(* CODESYS project LRF_2005_actual1.project
   Title: TemplateSPK1xxM01
   Version: 3.5.11.50
   Company: Production association OWEN

Project tree, tasks and I/O mapping:
  Device : SPK1xx[M01], Production association OWEN, order no. 7, version 3.5.11.57
    application Application
      libraries: Standard, * (System); CAA Memory, * (CAA Technical Workgroup); VisuDialogs, * (System); Standard64, * (System); VisuSymbols, 3.5.10.0 (System); Util, * (System)
      task OwenCloudTask (cyclic, interval T#100ms, priority 31) calls OwenStorage.CLOUD_PRG
      task MainTask (cyclic, interval t#10ms, priority 1) calls Main, Alarm, Motors
      task AlarmManagerTask (cyclic, interval 50 ms, priority 31) calls AlarmManager.Alarm_Prg
      task VISU_TASK (cyclic, interval 100 ms, priority 31) calls VisuElems.Visu_Prg
      Alarm Configuration
        alarm class Error (priority 10, acknowledge ACK_REP)
        alarm class Info (priority 100, acknowledge REP)
        alarm class Warning (priority 30, acknowledge REP)
        alarm group AlarmGroup
            11 [Error]: Comparison Equal, ExpressionToCompare TRUE, Expression GVL.SQ08_ALM - "Превышено время ожидания на переворот кантователя SQ08"
            21 [Error]: Comparison Equal, ExpressionToCompare TRUE, Expression GVL.M09UZ09_ALM - "Авария транспортера №5 M09UZ09"
            14 [Error]: Comparison Equal, ExpressionToCompare TRUE, Expression GVL.M01UZ01_ALM - "Авария дозатора обсыпного бункера M01UZ01"
            24 [Error]: Comparison Equal, ExpressionToCompare TRUE, Expression GVL.M14UZ14_ALM - "Авария транспортера №8 M14UZ14"
            19 [Error]: Comparison Equal, ExpressionToCompare TRUE, Expression GVL.M06UZ06_ALM - "Авария транспортера №3 M06UZ06"
            17 [Error]: Comparison Equal, ExpressionToCompare TRUE, Expression GVL.M04KM04_ALM - "Авария электромагнитного тормаза резчика M04KM04"
            12 [Info]: Comparison Equal, ExpressionToCompare TRUE, Expression GVL.XV01KV207_TSTOI - "Включен тестовый режим пресса "СЖАТЬ" XV01KV207"
            22 [Error]: Comparison Equal, ExpressionToCompare TRUE, Expression GVL.M11KM11_ALM - "Авария транспортера возврата песка №6 M11KM11"
            15 [Error]: Comparison Equal, ExpressionToCompare TRUE, Expression GVL.M02UZ02_ALM - "Авария резчика M02UZ02"
            25 [Error]: Comparison Equal, ExpressionToCompare TRUE, Expression GVL.A2_DI_SQ06_ALM - "Авария датчика верхнего положения выталкивателя SQ06 (геркон)."
            16 [Error]: Comparison Equal, ExpressionToCompare TRUE, Expression GVL.M03UZ03_ALM - "Авария транспортера №1 M03UZ03"
            10 [Error]: Comparison Equal, ExpressionToCompare TRUE, Expression GVL.M10KM10_ALM - "Авария маслостанции"
            20 [Error]: Comparison Equal, ExpressionToCompare TRUE, Expression GVL.M08KM08_ALM - "Авария транспортера подачи рамок №4 M08KM08"
            13 [Error]: Comparison Equal, ExpressionToCompare TRUE, Expression GVL.MV01KM00_ALM - "Авария вибратора обсыпного бункера MV01KM00"
            23 [Error]: Comparison Equal, ExpressionToCompare TRUE, Expression GVL.M12KM12_ALM - "Авария транспортера возврата обрези №7 M12KM12"
            18 [Error]: Comparison Equal, ExpressionToCompare TRUE, Expression GVL.M05UZ05_ALM - "Авария транспортера №2 M05UZ05"
            8 [Error]: Comparison Equal, ExpressionToCompare TRUE, Expression GVL.M07KM07_ALM - "Авария кантователя M07KM07"
            9 [Error]: Comparison Equal, ExpressionToCompare TRUE, Expression GVL.PI01_ALM - "Низкое давление масла PI01"
            0 [Error]: Comparison Equal, ExpressionToCompare FALSE, Expression GVL.A1_DI_SB_ALARM_STOP - "Нажата аварийная кнопка"
            1 [Error]: Comparison Equal, ExpressionToCompare TRUE, Expression GVL.A1_DI_QF25OK_ALM - "Отсутствует напряжение +24V QF25"
            2 [Error]: Comparison Equal, ExpressionToCompare TRUE, Expression GVL.A1_DI_QF26OK_ALM - "Отсутствует напряжение +24V QF26"
            3 [Error]: Comparison Equal, ExpressionToCompare TRUE, Expression GVL.A1_DI_380OK_ALM - "Отсутствует напряжение 380V QF1..QF16"
            4 [Error]: Comparison Equal, ExpressionToCompare TRUE, Expression GVL.XV01KV207_ALM - "Превышено время ожидания на сжатие пресса SQ05"
            5 [Error]: Comparison Equal, ExpressionToCompare TRUE, Expression GVL.XV02KV208_ALM - "Превышено время ожидания на разжатие пресса SQ04"
            6 [Error]: Comparison Equal, ExpressionToCompare TRUE, Expression GVL.XV03KV209_ALM - "Превышено время ожидания на выталкивание"
            7 [Error]: Comparison Equal, ExpressionToCompare TRUE, Expression GVL.XV04KV210_ALM - "Превышено время ожидания на возврат выталкивателя SQ06"
        text list AlarmGroup
        AlarmStorage
      global variables GVL
      visualisation TEST_FRAME_2
      program Motors [ST]
      visualisation SETTINGS_FRAME
      program SEQUENSER [ST]
      text list Mode
      visualisation PRF_FRAME
      TargetVariables/
        data type TRG_Drives
        data type TRG_Buzzer
        data type TRG_RTC
        global variables TargetVars
        data type TRG_Network
        data type TRG_Info
        data type TRG_Watchdog
        data type TRG_Debug
      visualisation ALARM_FRAME
      visualisation MODE_FRAME
      text list IM_TAGS
      visualisation TEST_FRAME_1
      visualisation Main
      program Alarm [ST]
      image pool Images
      program Main [ST]
      visualisation MAIN_FRAME
      text list IM
      visualisation MANUAL_FRAME_1
      global variables GVLR
      visualisation MANUAL_FRAME_2
      visualisation MANUAL_FRAME_3
    Info : Info, Production association OWEN, version 3.5.11.5003
        input  Application.TargetVars.stInfo.sVendorName : ARRAY [0..80] OF BYTE  // VENDOR
        input  Application.TargetVars.stInfo.sDeviceName : ARRAY [0..80] OF BYTE  // DEVICE
        input  Application.TargetVars.stInfo.sSerialId : ARRAY [0..80] OF BYTE  // SERIAL
        input  Application.TargetVars.stInfo.sRuntimeVersion : ARRAY [0..80] OF BYTE  // RUNTIME
        input  Application.TargetVars.stInfo.sFirmwareVersion : ARRAY [0..80] OF BYTE  // FIRMWARE
        input  Application.TargetVars.stInfo.sLinuxVersion : ARRAY [0..80] OF BYTE  // LINUX
        input  Application.TargetVars.stInfo.sNeedTargetVersion : ARRAY [0..80] OF BYTE  // TARGET
        input  Application.TargetVars.stInfo.sProjectName : ARRAY [0..80] OF BYTE  // PROJECT
        input  Application.TargetVars.stInfo.sAuthorName : ARRAY [0..80] OF BYTE  // AUTHOR
        input  Application.TargetVars.stInfo.sProjectVersion : ARRAY [0..80] OF BYTE  // VERSION
        input  Application.TargetVars.stInfo.sProjectProfile : ARRAY [0..80] OF BYTE  // PROFILE
        input  Application.TargetVars.stInfo.dtProjectLastChanges : DT  // LASTCHANGES
    Drives : Drives, Production association OWEN, version 3.5.11.5002
        input  Application.TargetVars.stDrives.uliFsFullSize : ULINT  // FS size
        input  Application.TargetVars.stDrives.uliFsUsedSize : ULINT  // FS used
        input  Application.TargetVars.stDrives.uliFsFreeSize : ULINT  // FS free
        input  Application.TargetVars.stDrives.xUsbMounted : BIT  // USB Mounted
        input  Application.TargetVars.stDrives.xUsbUnmountDone : BIT  // USB Unmount done
        input  Application.TargetVars.stDrives.uliUsbFullSize : ULINT  // USB size
        input  Application.TargetVars.stDrives.uliUsbUsedSize : ULINT  // USB used
        input  Application.TargetVars.stDrives.uliUsbFreeSize : ULINT  // USB free
        input  Application.TargetVars.stDrives.xSdMounted : BIT  // MMC Mounted
        input  Application.TargetVars.stDrives.xSdUnmountDone : BIT  // MMC Unmount done
        input  Application.TargetVars.stDrives.uliSdFullSize : ULINT  // MMC size
        input  Application.TargetVars.stDrives.uliSdUsedSize : ULINT  // MMC used
        input  Application.TargetVars.stDrives.uliSdFreeSize : ULINT  // MMC free
        output Application.TargetVars.stDrives.xEnable : BIT  // Enable Drives
        output Application.TargetVars.stDrives.xUsbUnmount : BIT  // USB Unmount
        output Application.TargetVars.stDrives.xSdUnmount : BIT  // MMC Unmount
    RS232_2 : Modbus COM, 3S - Smart Software Solutions GmbH, version 3.5.11.20
        settings: DataBits = 8; StopBits = 1; ComPort = 5
    OwenRTC : OwenRTC, Production association OWEN, version 3.5.11.5003
        input  Application.TargetVars.stRtc.uiGetYear : UINT  // Year
        input  Application.TargetVars.stRtc.usiGetMonth : USINT  // Month
        input  Application.TargetVars.stRtc.usiGetDay : USINT  // Day
        input  Application.TargetVars.stRtc.usiGetHour : USINT  // Hour
        input  Application.TargetVars.stRtc.usiGetMinute : USINT  // Minute
        input  Application.TargetVars.stRtc.usiGetSecond : USINT  // Second
        input  Application.TargetVars.stRtc.usiGetDayOfWeek : USINT  // Day of Week
        input  Application.TargetVars.stRtc.usiGetWeekOfYear : USINT  // Week of Year
        input  Application.GVL.PLC_DATE : ARRAY [0..80] OF BYTE  // Format Date
        input  Application.GVL.PLC_TIME : ARRAY [0..80] OF BYTE  // Format Time
        input  Application.TargetVars.stRtc.siGetUtcOffset : SINT  // UTC Offset
        input  Application.TargetVars.stRtc.xIsNtpEnabled : BIT  // NTP Enabled
        input  Application.TargetVars.stRtc.usiNtpErrorCode : USINT  // NTP Error
        input  Application.TargetVars.stRtc.ltSystemTick : LTIME  // System Timer
        input  Application.TargetVars.stRtc.dtDateAndTime : DT  // Date And Time
        output Application.TargetVars.stRtc.uiSetYear : UINT  // New Year
        output Application.TargetVars.stRtc.usiSetMonth : USINT  // New Month
        output Application.TargetVars.stRtc.usiSetDay : USINT  // New Day
        output Application.TargetVars.stRtc.usiSetHour : USINT  // New Hour
        output Application.TargetVars.stRtc.usiSetMinute : USINT  // New Minute
        output Application.TargetVars.stRtc.usiSetSecond : USINT  // New Second
        output Application.TargetVars.stRtc.siSetUtcOffset : SINT  // New UTC Offset
        output Application.TargetVars.stRtc.xUpdateSettings : BIT  // Set Settings DT
        output Application.TargetVars.stRtc.xEnableNtp : BIT  // Enable NTP
        output Application.TargetVars.stRtc.sPreferNtpServer : ARRAY [0..80] OF BYTE  // Prefer Server
    Debug : Debug, Production association OWEN, version 3.5.11.5002
        input  Application.TargetVars.stDebug.udiRamUsedSize : UDINT  // RAM used
        input  Application.TargetVars.stDebug.udiRamFreeSize : UDINT  // RAM free
        input  Application.TargetVars.stDebug.udiCountHandles : UDINT  // Open files
        input  Application.TargetVars.stDebug.udiProcUsage : UDINT  // Processor usage
        output Application.TargetVars.stDebug.xEnable : BIT  // Enable Debug
        output Application.TargetVars.stDebug.udiPollingTime : UDINT  // Debug pause
        unmapped channels: Core temp
    Watchdog : Watchdog, Production association OWEN, version 3.5.11.5003
        input  Application.TargetVars.stWatchdog.eHandlingType : INT  // Exception Handling
        input  Application.TargetVars.stWatchdog.udiLastExceptionCode : UDINT  // Last Exception Code
        input  Application.TargetVars.stWatchdog.sLastExceptionText : localTypes:STRING  // Last Exception Description
        input  Application.TargetVars.stWatchdog.dtLastExceptionTime : DT  // Last Exception Time
        input  Application.TargetVars.stWatchdog.xIsHardwareWatchdogReboot : BIT  // Hardware Watchdog Flag
        input  Application.TargetVars.stWatchdog.usiPowerRebootCount : USINT  // Power Reboot Count
        input  Application.TargetVars.stWatchdog.usiHardwareWatchdogRebootCount : USINT  // Watchdog Reboot Count
        input  Application.TargetVars.stWatchdog.usiExceptionRebootCount : USINT  // Exception Reboot Count
        input  Application.TargetVars.stWatchdog.usiCommandRebootCount : USINT  // Command Reboot Count
        output Application.TargetVars.stWatchdog.xDoReboot : BIT  // Reboot
        output Application.TargetVars.stWatchdog.xResetCounters : BIT  // Reset Counters
    Ethernet : Ethernet, 3S - Smart Software Solutions GmbH, version 3.5.11.0
        settings: IPAddress = [192,168,0,10]; SubnetMask = [255,255,0,0]; GatewayAddress = [192,168,0,1]; MACAddress = [16#E4,16#1E,16#0A,16#00,16#8E,16#B8]; NetworkInterfaceName = 'eth0'; NetworkInterfaceName = "eth0"; SaveCommunicationSettings = FALSE
      Modbus_TCP_Master : Modbus TCP Master, 3S - Smart Software Solutions GmbH, version 3.5.11.30
        A4 : MU210-410, Production association OWEN, version 3.5.11.6
            settings: IPAddress = [192, 168, 0, 6]
            input  Application.GVL.A4_DI_Modul_Fail : BIT  // Флаг ошибки
            output Application.GVL.A4_DO_HL02_32 : BOOL  // Битовая маска выходов (запись).Выход 1
            output Application.GVL.A4_DO_HL21 : BOOL  // Битовая маска выходов (запись).Выход 2
            output Application.GVL.A4_DO_HL35 : BOOL  // Битовая маска выходов (запись).Выход 3
            output Application.GVL.A4_DO_HL03_33 : BOOL  // Битовая маска выходов (запись).Выход 4
            output Application.GVL.A4_DO_HL04_34 : BOOL  // Битовая маска выходов (запись).Выход 5
            output Application.GVL.A4_DO_HL05 : BOOL  // Битовая маска выходов (запись).Выход 6
            output Application.GVL.A4_DO_XV01KV207 : BOOL  // Битовая маска выходов (запись).Выход 7
            output Application.GVL.A4_DO_XV02KV208 : BOOL  // Битовая маска выходов (запись).Выход 8
            output Application.GVL.A4_DO_XV03KV209 : BOOL  // Битовая маска выходов (запись).Выход 9
            output Application.GVL.A4_DO_XV04KV210 : BOOL  // Битовая маска выходов (запись).Выход 10
            output Application.GVL.A4_DO_XV05KV211 : BOOL  // Битовая маска выходов (запись).Выход 11
            output Application.GVL.A4_DO_XV06KV212 : BOOL  // Битовая маска выходов (запись).Выход 12
            output Application.GVL.A4_DO_RESERV01 : BOOL  // Битовая маска выходов (запись).Выход 13
            output Application.GVL.A4_DO_RESERV02 : BOOL  // Битовая маска выходов (запись).Выход 14
            output Application.GVL.A5_DO_M02UZ02_RUN_REV : BOOL  // Битовая маска выходов (запись).Выход 15
            output Application.GVL.A4_DO_RESERV04 : BOOL  // Битовая маска выходов (запись).Выход 16
            unmapped channels: Tmp, Исключить модуль из опроса, Битовая маска выходов (чтение), Битовая маска выходов (запись), Битовая маска диагностики выходов, Параметр ШИМ (чтение), Параметр ШИМ (чтение), Параметр ШИМ (чтение), Параметр ШИМ (чтение), Параметр ШИМ (чтение), Параметр ШИМ (чтение), Параметр ШИМ (чтение), Параметр ШИМ (чтение), Период ШИМ (чтение), Период ШИМ (чтение), Период ШИМ (чтение), Период ШИМ (чтение), Период ШИМ (чтение), Период ШИМ (чтение), Период ШИМ (чтение), Период ШИМ (чтение), Параметр ШИМ (запись), Параметр ШИМ (запись), Параметр ШИМ (запись), Параметр ШИМ (запись), Параметр ШИМ (запись), Параметр ШИМ (запись), Параметр ШИМ (запись), Параметр ШИМ (запись), Период ШИМ (запись), Период ШИМ (запись), Период ШИМ (запись), Период ШИМ (запись), Период ШИМ (запись), Период ШИМ (запись), Период ШИМ (запись), Период ШИМ (запись), Коэффициент заполнения ШИМ (чтение), Коэффициент заполнения ШИМ (чтение), Коэффициент заполнения ШИМ (чтение),
              Коэффициент заполнения ШИМ (чтение), Коэффициент заполнения ШИМ (чтение), Коэффициент заполнения ШИМ (чтение), Коэффициент заполнения ШИМ (чтение), Коэффициент заполнения ШИМ (чтение), Коэффициент заполнения ШИМ (чтение), Коэффициент заполнения ШИМ (чтение), Коэффициент заполнения ШИМ (чтение), Коэффициент заполнения ШИМ (чтение), Коэффициент заполнения ШИМ (чтение), Коэффициент заполнения ШИМ (чтение), Коэффициент заполнения ШИМ (чтение), Коэффициент заполнения ШИМ (чтение), Коэффициент заполнения ШИМ (запись), Коэффициент заполнения ШИМ (запись), Коэффициент заполнения ШИМ (запись), Коэффициент заполнения ШИМ (запись), Коэффициент заполнения ШИМ (запись), Коэффициент заполнения ШИМ (запись), Коэффициент заполнения ШИМ (запись), Коэффициент заполнения ШИМ (запись), Коэффициент заполнения ШИМ (запись), Коэффициент заполнения ШИМ (запись), Коэффициент заполнения ШИМ (запись), Коэффициент заполнения ШИМ (запись), Коэффициент заполнения ШИМ (запись), Коэффициент заполнения ШИМ (запись), Коэффициент заполнения ШИМ (запись), Коэффициент заполнения ШИМ (запись), Прочитать параметры, Записать параметры, Записать параметры, Записать параметры, Частота генератора (чтение), Частота генератора (чтение), Частота генератора (чтение), Частота генератора (запись), Частота генератора (запись), Частота генератора (запись), Количество импульсов генератора (чтение),
              Количество импульсов генератора (чтение), Количество импульсов генератора (чтение), Количество импульсов генератора (запись), Количество импульсов генератора (запись), Количество импульсов генератора (запись), Осталось сгенерировать импульсов, Осталось сгенерировать импульсов, Осталось сгенерировать импульсов
        A1 : MV210-202, Production association OWEN, version 3.5.11.6
            settings: IPAddress = [192, 168, 0, 3]
            input  Application.GVL.A1_DI_Modul_Fail : BIT  // Флаг ошибки
            input  Application.GVL.A1_DI_QF25OK : BOOL  // Битовая маска входов.Вход 1
            input  Application.GVL.A1_DI_QF26OK : BOOL  // Битовая маска входов.Вход 2
            input  Application.GVL.A1_DI_380OK : BOOL  // Битовая маска входов.Вход 3
            input  Application.GVL.A1_DI_SB_ALARM_STOP : BOOL  // Битовая маска входов.Вход 4
            input  Application.GVL.A1_DI_SB_STOP : BOOL  // Битовая маска входов.Вход 5
            input  Application.GVL.A1_DI_SB_1st_OPER : BOOL  // Битовая маска входов.Вход 6
            input  Application.GVL.A1_DI_SB_2nd_OPER : BOOL  // Битовая маска входов.Вход 7
            input  Application.GVL.A1_DI_SB_RESET : BOOL  // Битовая маска входов.Вход 8
            input  Application.GVL.A1_DI_SB_START : BOOL  // Битовая маска входов.Вход 9
            input  Application.GVL.A1_DI_SA01 : BOOL  // Битовая маска входов.Вход 10
            input  Application.GVL.A1_DI_SB_TEST : BOOL  // Битовая маска входов.Вход 11
            input  Application.GVL.A1_DI_MV01KM00_ON : BOOL  // Битовая маска входов.Вход 12
            input  Application.GVL.A1_DI_M01UZ01_ON : BOOL  // Битовая маска входов.Вход 13
            input  Application.GVL.A1_DI_RESERV01 : BOOL  // Битовая маска входов.Вход 14
            input  Application.GVL.A1_DI_M03UZ03_ON : BOOL  // Битовая маска входов.Вход 15
            input  Application.GVL.A1_DI_M04KM04_ON : BOOL  // Битовая маска входов.Вход 16
            input  Application.GVL.A1_DI_M05UZ05_ON : BOOL  // Битовая маска входов.Вход 17
            input  Application.GVL.A1_DI_M06UZ06_ON : BOOL  // Битовая маска входов.Вход 18
            input  Application.GVL.A1_DI_M07KM07_ON : BOOL  // Битовая маска входов.Вход 19
            input  Application.GVL.A1_DI_M08KM08_ON : BOOL  // Битовая маска входов.Вход 20
            unmapped channels: Tmp, Исключить модуль из опроса, Битовая маска входов, Значение, Значение, Значение, Значение, Значение, Значение, Значение, Значение, Значение счетчика, Значение счетчика, Значение счетчика, Значение счетчика, Значение счетчика, Значение счетчика, Значение счетчика, Значение счетчика, Значение счетчика, Значение счетчика, Значение счетчика, Значение счетчика, Сбросить значение, Сбросить значение, Сбросить значение, Сбросить значение, Сбросить значение, Сбросить значение, Сбросить значение, Сбросить значение, Сбросить счетчик, Сбросить счетчик, Сбросить счетчик, Сбросить счетчик, Сбросить счетчик, Сбросить счетчик, Сбросить счетчик, Сбросить счетчик, Сбросить счетчик,
              Сбросить счетчик, Сбросить счетчик, Сбросить счетчик
        A5 : MU210-410, Production association OWEN, version 3.5.11.6
            settings: IPAddress = [192, 168, 0, 7]
            input  Application.GVL.A5_DI_Modul_Fail : BIT  // Флаг ошибки
            output Application.GVL.A5_DO_MV01KM00_RUN : BOOL  // Битовая маска выходов (запись).Выход 1
            output Application.GVL.A5_DO_M01UZ01_RUN : BOOL  // Битовая маска выходов (запись).Выход 2
            output Application.GVL.A5_DO_M02UZ02_RUN_FORW : BOOL  // Битовая маска выходов (запись).Выход 3
            output Application.GVL.A5_DO_M03UZ03_RUN : BOOL  // Битовая маска выходов (запись).Выход 4
            output Application.GVL.A5_DO_M04KM04_RUN : BOOL  // Битовая маска выходов (запись).Выход 5
            output Application.GVL.A5_DO_M05UZ05_RUN : BOOL  // Битовая маска выходов (запись).Выход 6
            output Application.GVL.A5_DO_M06UZ06_RUN : BOOL  // Битовая маска выходов (запись).Выход 7
            output Application.GVL.A5_DO_M07KM07_RUN : BOOL  // Битовая маска выходов (запись).Выход 8
            output Application.GVL.A5_DO_M08KM08_RUN : BOOL  // Битовая маска выходов (запись).Выход 9
            output Application.GVL.A5_DO_M09UZ09_RUN : BOOL  // Битовая маска выходов (запись).Выход 10
            output Application.GVL.A5_DO_M10KM10_RUN : BOOL  // Битовая маска выходов (запись).Выход 11
            output Application.GVL.A5_DO_M11KM11_RUN : BOOL  // Битовая маска выходов (запись).Выход 12
            output Application.GVL.A5_DO_M12KM12_RUN : BOOL  // Битовая маска выходов (запись).Выход 13
            output Application.GVL.A5_DO_M13KM13_RUN : BOOL  // Битовая маска выходов (запись).Выход 14
            output Application.GVL.A5_DO_M14UZ14_RUN : BOOL  // Битовая маска выходов (запись).Выход 15
            output Application.GVL.A5_DO_RESERV01 : BOOL  // Битовая маска выходов (запись).Выход 16
            unmapped channels: Tmp, Исключить модуль из опроса, Битовая маска выходов (чтение), Битовая маска выходов (запись), Битовая маска диагностики выходов, Параметр ШИМ (чтение), Параметр ШИМ (чтение), Параметр ШИМ (чтение), Параметр ШИМ (чтение), Параметр ШИМ (чтение), Параметр ШИМ (чтение), Параметр ШИМ (чтение), Параметр ШИМ (чтение), Период ШИМ (чтение), Период ШИМ (чтение), Период ШИМ (чтение), Период ШИМ (чтение), Период ШИМ (чтение), Период ШИМ (чтение), Период ШИМ (чтение), Период ШИМ (чтение), Параметр ШИМ (запись), Параметр ШИМ (запись), Параметр ШИМ (запись), Параметр ШИМ (запись), Параметр ШИМ (запись), Параметр ШИМ (запись), Параметр ШИМ (запись), Параметр ШИМ (запись), Период ШИМ (запись), Период ШИМ (запись), Период ШИМ (запись), Период ШИМ (запись), Период ШИМ (запись), Период ШИМ (запись), Период ШИМ (запись), Период ШИМ (запись), Коэффициент заполнения ШИМ (чтение), Коэффициент заполнения ШИМ (чтение), Коэффициент заполнения ШИМ (чтение),
              Коэффициент заполнения ШИМ (чтение), Коэффициент заполнения ШИМ (чтение), Коэффициент заполнения ШИМ (чтение), Коэффициент заполнения ШИМ (чтение), Коэффициент заполнения ШИМ (чтение), Коэффициент заполнения ШИМ (чтение), Коэффициент заполнения ШИМ (чтение), Коэффициент заполнения ШИМ (чтение), Коэффициент заполнения ШИМ (чтение), Коэффициент заполнения ШИМ (чтение), Коэффициент заполнения ШИМ (чтение), Коэффициент заполнения ШИМ (чтение), Коэффициент заполнения ШИМ (чтение), Коэффициент заполнения ШИМ (запись), Коэффициент заполнения ШИМ (запись), Коэффициент заполнения ШИМ (запись), Коэффициент заполнения ШИМ (запись), Коэффициент заполнения ШИМ (запись), Коэффициент заполнения ШИМ (запись), Коэффициент заполнения ШИМ (запись), Коэффициент заполнения ШИМ (запись), Коэффициент заполнения ШИМ (запись), Коэффициент заполнения ШИМ (запись), Коэффициент заполнения ШИМ (запись), Коэффициент заполнения ШИМ (запись), Коэффициент заполнения ШИМ (запись), Коэффициент заполнения ШИМ (запись), Коэффициент заполнения ШИМ (запись), Коэффициент заполнения ШИМ (запись), Прочитать параметры, Записать параметры, Записать параметры, Записать параметры, Частота генератора (чтение), Частота генератора (чтение), Частота генератора (чтение), Частота генератора (запись), Частота генератора (запись), Частота генератора (запись), Количество импульсов генератора (чтение),
              Количество импульсов генератора (чтение), Количество импульсов генератора (чтение), Количество импульсов генератора (запись), Количество импульсов генератора (запись), Количество импульсов генератора (запись), Осталось сгенерировать импульсов, Осталось сгенерировать импульсов, Осталось сгенерировать импульсов
        A3 : MK210-302, Production association OWEN, version 3.5.11.6
            settings: IPAddress = [192, 168, 0, 5]
            input  Application.GVL.A3_DI_Modul_Fail : BIT  // Флаг ошибки
            input  Application.GVL.A3_DI_SQ10 : BOOL  // Битовая маска входов.Вход 1
            input  Application.GVL.A3_DI_SQ13 : BOOL  // Битовая маска входов.Вход 2
            input  Application.GVL.A3_DI_SQ14 : BOOL  // Битовая маска входов.Вход 3
            input  Application.GVL.A3_DI_RESERV01 : BOOL  // Битовая маска входов.Вход 4
            input  Application.GVL.A3_DI_SQ11 : BOOL  // Битовая маска входов.Вход 5
            input  Application.GVL.A3_DI_SQ12 : BOOL  // Битовая маска входов.Вход 6
            input  Application.GVL.A3_DI_RESERV02 : BOOL  // Битовая маска входов.Вход 7
            input  Application.GVL.A3_DI_KV301 : BOOL  // Битовая маска входов.Вход 8
            input  Application.GVL.A3_DI_KV302 : BOOL  // Битовая маска входов.Вход 9
            input  Application.GVL.A3_DI_PI01 : BOOL  // Битовая маска входов.Вход 10
            input  Application.GVL.A3_DI_RESERV03 : BOOL  // Битовая маска входов.Вход 11
            input  Application.GVL.A3_DI_RESERV04 : BOOL  // Битовая маска входов.Вход 12
            output Application.GVL.A3_DO_KV303 : BOOL  // Битовая маска выходов (запись).Выход 1
            output Application.GVL.A3_DO_KV304 : BOOL  // Битовая маска выходов (запись).Выход 2
            output Application.GVL.A3_DO_RESERV01 : BOOL  // Битовая маска выходов (запись).Выход 3
            output Application.GVL.A3_DO_RESERV02 : BOOL  // Битовая маска выходов (запись).Выход 4
            unmapped channels: Tmp, Исключить модуль из опроса, Битовая маска входов, Значение счетчика, Значение счетчика, Значение счетчика, Значение счетчика, Значение счетчика, Значение счетчика, Значение счетчика, Значение счетчика, Значение счетчика, Значение счетчика, Значение счетчика, Значение счетчика, Битовая маска выходов (чтение), Битовая маска выходов (запись), Сбросить счетчик, Сбросить счетчик, Сбросить счетчик, Сбросить счетчик, Сбросить счетчик, Сбросить счетчик, Сбросить счетчик, Сбросить счетчик, Сбросить счетчик, Сбросить счетчик, Сбросить счетчик, Сбросить счетчик, Период ШИМ (чтение), Период ШИМ (чтение), Период ШИМ (чтение), Период ШИМ (чтение), Период ШИМ (запись), Период ШИМ (запись), Период ШИМ (запись), Период ШИМ (запись), Коэффициент заполнения ШИМ (чтение), Коэффициент заполнения ШИМ (чтение), Коэффициент заполнения ШИМ (чтение),
              Коэффициент заполнения ШИМ (чтение), Коэффициент заполнения ШИМ (запись), Коэффициент заполнения ШИМ (запись), Коэффициент заполнения ШИМ (запись), Коэффициент заполнения ШИМ (запись)
        A2 : MV210-202, Production association OWEN, version 3.5.11.6
            settings: IPAddress = [192, 168, 0, 4]
            input  Application.GVL.A2_DI_Modul_Fail : BIT  // Флаг ошибки
            input  Application.GVL.A2_DI_M09UZ09_ON : BOOL  // Битовая маска входов.Вход 1
            input  Application.GVL.A2_DI_M10KM10_ON : BOOL  // Битовая маска входов.Вход 2
            input  Application.GVL.A2_DI_M11KM11_ON : BOOL  // Битовая маска входов.Вход 3
            input  Application.GVL.A2_DI_M12KM12_ON : BOOL  // Битовая маска входов.Вход 4
            input  Application.GVL.A2_DI_M13KM13_ON : BOOL  // Битовая маска входов.Вход 5
            input  Application.GVL.A2_DI_M14UZ14_ON : BOOL  // Битовая маска входов.Вход 6
            input  Application.GVL.A2_DI_SQ01 : BOOL  // Битовая маска входов.Вход 7
            input  Application.GVL.A2_DI_SQ02 : BOOL  // Битовая маска входов.Вход 8
            input  Application.GVL.A2_DI_SQ15 : BOOL  // Битовая маска входов.Вход 9
            input  Application.GVL.A2_DI_SQ03 : BOOL  // Битовая маска входов.Вход 10
            input  Application.GVL.A2_DI_RESERV02 : BOOL  // Битовая маска входов.Вход 11
            input  Application.GVL.A2_DI_SQ04 : BOOL  // Битовая маска входов.Вход 12
            input  Application.GVL.A2_DI_SQ05 : BOOL  // Битовая маска входов.Вход 13
            input  Application.GVL.A2_DI_SQ06 : BOOL  // Битовая маска входов.Вход 14
            input  Application.GVL.A2_DI_SQ07 : BOOL  // Битовая маска входов.Вход 15
            input  Application.GVL.A2_DI_SQ08 : BOOL  // Битовая маска входов.Вход 16
            input  Application.GVL.A2_DI_RESERV03 : BOOL  // Битовая маска входов.Вход 17
            input  Application.GVL.A2_DI_RESERV04 : BOOL  // Битовая маска входов.Вход 18
            input  Application.GVL.A2_DI_RESERV05 : BOOL  // Битовая маска входов.Вход 19
            input  Application.GVL.A2_DI_SQ09 : BOOL  // Битовая маска входов.Вход 20
            input  Application.GVL.A2_DI_SQ02_CNT : UDINT  // Значение
            input  Application.GVL.A2_DI_SQ08_CNT : UDINT  // Значение счетчика
            output Application.GVL.RESET_SQ2_CNT : BIT  // Сбросить значение
            output Application.GVL.RESET_CNT : BIT  // Сбросить счетчик
            unmapped channels: Tmp, Исключить модуль из опроса, Битовая маска входов, Значение, Значение, Значение, Значение, Значение, Значение, Значение, Значение счетчика, Значение счетчика, Значение счетчика, Значение счетчика, Значение счетчика, Значение счетчика, Значение счетчика, Значение счетчика, Значение счетчика, Значение счетчика, Значение счетчика, Сбросить значение, Сбросить значение, Сбросить значение, Сбросить значение, Сбросить значение, Сбросить значение, Сбросить значение, Сбросить счетчик, Сбросить счетчик, Сбросить счетчик, Сбросить счетчик, Сбросить счетчик, Сбросить счетчик, Сбросить счетчик, Сбросить счетчик, Сбросить счетчик, Сбросить счетчик, Сбросить счетчик
    RS485_2 : Modbus COM, 3S - Smart Software Solutions GmbH, version 3.5.11.20
        settings: DataBits = 8; StopBits = 1; ComPort = 2
    RS485_3 : Modbus COM, 3S - Smart Software Solutions GmbH, version 3.5.11.20
        settings: DataBits = 8; StopBits = 1; ComPort = 3
    RS232_1 : Modbus COM, 3S - Smart Software Solutions GmbH, version 3.5.11.20
        settings: DataBits = 8; StopBits = 1; ComPort = 4
    RS485_1 : Modbus COM, 3S - Smart Software Solutions GmbH, version 3.5.11.20
        settings: DataBits = 8; StopBits = 1; ComPort = 1
      Modbus_Master_COM_Port_1 : Modbus Master, COM Port, 3S - Smart Software Solutions GmbH, version 3.5.11.20
        UZ06 : Modbus Slave, COM Port, 3S - Smart Software Solutions GmbH, version 3.5.10.30
            settings: SlaveAddress = 6; ResponseTimeout = 1000; UseExtendedFunctionCodes = TRUE; UZ_FREQUENCY_PV.Function Code = 3; UZ_FREQUENCY_PV.Read Offset = 16#C421; UZ_FREQUENCY_PV.Read Length = 1; UZ_FREQUENCY_PV.Write Offset = 0; UZ_FREQUENCY_PV.Write Length = 0; UZ_FREQUENCY_PV.Cycle Time = 100; UZ_STATUS.Function Code = 3; UZ_STATUS.Read Offset = 16#C417; UZ_STATUS.Read Length = 1; UZ_STATUS.Write Offset = 0; UZ_STATUS.Write Length = 0; UZ_STATUS.Cycle Time = 100; UZ_CONTROL.Function Code = 6; UZ_CONTROL.Read Offset = 0; UZ_CONTROL.Read Length = 0; UZ_CONTROL.Write Offset = 16#C34F; UZ_CONTROL.Write Length = 1; UZ_CONTROL.Cycle Time = 100; UZ_FREQUENCY_SP.Function Code = 6; UZ_FREQUENCY_SP.Read Offset = 0; UZ_FREQUENCY_SP.Read Length = 0; UZ_FREQUENCY_SP.Write Offset = 16#C359; UZ_FREQUENCY_SP.Write Length = 1; UZ_FREQUENCY_SP.Cycle Time = 100
            input  Application.GVL.UZ06_Freq_PV : ARRAY[0..0] OF WORD  // UZ_FREQUENCY_PV
            output Application.GVL.UZ06_Freq_SP : ARRAY[0..0] OF WORD  // UZ_FREQUENCY_SP
            unmapped channels: UZ_STATUS, UZ_CONTROL
        UZ03 : Modbus Slave, COM Port, 3S - Smart Software Solutions GmbH, version 3.5.10.30
            settings: SlaveAddress = 3; ResponseTimeout = 1000; UseExtendedFunctionCodes = TRUE; UZ_FREQUENCY_PV.Function Code = 3; UZ_FREQUENCY_PV.Read Offset = 16#C421; UZ_FREQUENCY_PV.Read Length = 1; UZ_FREQUENCY_PV.Write Offset = 0; UZ_FREQUENCY_PV.Write Length = 0; UZ_FREQUENCY_PV.Cycle Time = 100; UZ_STATUS.Function Code = 3; UZ_STATUS.Read Offset = 16#C417; UZ_STATUS.Read Length = 1; UZ_STATUS.Write Offset = 0; UZ_STATUS.Write Length = 0; UZ_STATUS.Cycle Time = 100; UZ_CONTROL.Function Code = 6; UZ_CONTROL.Read Offset = 0; UZ_CONTROL.Read Length = 0; UZ_CONTROL.Write Offset = 16#C34F; UZ_CONTROL.Write Length = 1; UZ_CONTROL.Cycle Time = 100; UZ_FREQUENCY_SP.Function Code = 6; UZ_FREQUENCY_SP.Read Offset = 0; UZ_FREQUENCY_SP.Read Length = 0; UZ_FREQUENCY_SP.Write Offset = 16#C359; UZ_FREQUENCY_SP.Write Length = 1; UZ_FREQUENCY_SP.Cycle Time = 100
            input  Application.GVL.UZ03_Freq_PV : ARRAY[0..0] OF WORD  // UZ_FREQUENCY_PV
            input  Application.GVL.UZ03_Status_Word : ARRAY[0..0] OF WORD  // UZ_STATUS
            output Application.GVL.UZ03_Freq_SP : ARRAY[0..0] OF WORD  // UZ_FREQUENCY_SP
            unmapped channels: UZ_CONTROL
        UZ05 : Modbus Slave, COM Port, 3S - Smart Software Solutions GmbH, version 3.5.10.30
            settings: SlaveAddress = 5; ResponseTimeout = 1000; UseExtendedFunctionCodes = TRUE; UZ_FREQUENCY_PV.Function Code = 3; UZ_FREQUENCY_PV.Read Offset = 16#C421; UZ_FREQUENCY_PV.Read Length = 1; UZ_FREQUENCY_PV.Write Offset = 0; UZ_FREQUENCY_PV.Write Length = 0; UZ_FREQUENCY_PV.Cycle Time = 100; UZ_STATUS.Function Code = 3; UZ_STATUS.Read Offset = 16#C417; UZ_STATUS.Read Length = 1; UZ_STATUS.Write Offset = 0; UZ_STATUS.Write Length = 0; UZ_STATUS.Cycle Time = 100; UZ_CONTROL.Function Code = 6; UZ_CONTROL.Read Offset = 0; UZ_CONTROL.Read Length = 0; UZ_CONTROL.Write Offset = 16#C34F; UZ_CONTROL.Write Length = 1; UZ_CONTROL.Cycle Time = 100; UZ_FREQUENCY_SP.Function Code = 6; UZ_FREQUENCY_SP.Read Offset = 0; UZ_FREQUENCY_SP.Read Length = 0; UZ_FREQUENCY_SP.Write Offset = 16#C359; UZ_FREQUENCY_SP.Write Length = 1; UZ_FREQUENCY_SP.Cycle Time = 100
            input  Application.GVL.UZ05_Freq_PV : ARRAY[0..0] OF WORD  // UZ_FREQUENCY_PV
            output Application.GVL.UZ05_Freq_SP : ARRAY[0..0] OF WORD  // UZ_FREQUENCY_SP
            unmapped channels: UZ_STATUS, UZ_CONTROL
        UZ09 : Modbus Slave, COM Port, 3S - Smart Software Solutions GmbH, version 3.5.10.30
            settings: SlaveAddress = 9; ResponseTimeout = 1000; UseExtendedFunctionCodes = TRUE; UZ_FREQUENCY_PV.Function Code = 3; UZ_FREQUENCY_PV.Read Offset = 16#C421; UZ_FREQUENCY_PV.Read Length = 1; UZ_FREQUENCY_PV.Write Offset = 0; UZ_FREQUENCY_PV.Write Length = 0; UZ_FREQUENCY_PV.Cycle Time = 100; UZ_STATUS.Function Code = 3; UZ_STATUS.Read Offset = 16#C417; UZ_STATUS.Read Length = 1; UZ_STATUS.Write Offset = 0; UZ_STATUS.Write Length = 0; UZ_STATUS.Cycle Time = 100; UZ_CONTROL.Function Code = 6; UZ_CONTROL.Read Offset = 0; UZ_CONTROL.Read Length = 0; UZ_CONTROL.Write Offset = 16#C34F; UZ_CONTROL.Write Length = 1; UZ_CONTROL.Cycle Time = 100; UZ_FREQUENCY_SP.Function Code = 6; UZ_FREQUENCY_SP.Read Offset = 0; UZ_FREQUENCY_SP.Read Length = 0; UZ_FREQUENCY_SP.Write Offset = 16#C359; UZ_FREQUENCY_SP.Write Length = 1; UZ_FREQUENCY_SP.Cycle Time = 100
            input  Application.GVL.UZ09_Freq_PV : ARRAY[0..0] OF WORD  // UZ_FREQUENCY_PV
            output Application.GVL.UZ09_Freq_SP : ARRAY[0..0] OF WORD  // UZ_FREQUENCY_SP
            unmapped channels: UZ_STATUS, UZ_CONTROL
        UZ02 : Modbus Slave, COM Port, 3S - Smart Software Solutions GmbH, version 3.5.10.30
            settings: SlaveAddress = 2; ResponseTimeout = 1000; UseExtendedFunctionCodes = TRUE; UZ_FREQUENCY_PV.Function Code = 3; UZ_FREQUENCY_PV.Read Offset = 16#C421; UZ_FREQUENCY_PV.Read Length = 1; UZ_FREQUENCY_PV.Write Offset = 0; UZ_FREQUENCY_PV.Write Length = 0; UZ_FREQUENCY_PV.Cycle Time = 100; UZ_STATUS.Function Code = 3; UZ_STATUS.Read Offset = 16#C417; UZ_STATUS.Read Length = 1; UZ_STATUS.Write Offset = 0; UZ_STATUS.Write Length = 0; UZ_STATUS.Cycle Time = 100; UZ_CONTROL.Function Code = 6; UZ_CONTROL.Read Offset = 0; UZ_CONTROL.Read Length = 0; UZ_CONTROL.Write Offset = 16#C34F; UZ_CONTROL.Write Length = 1; UZ_CONTROL.Cycle Time = 100; UZ_FREQUENCY_SP.Function Code = 6; UZ_FREQUENCY_SP.Read Offset = 0; UZ_FREQUENCY_SP.Read Length = 0; UZ_FREQUENCY_SP.Write Offset = 16#C359; UZ_FREQUENCY_SP.Write Length = 1; UZ_FREQUENCY_SP.Cycle Time = 100
            input  Application.GVL.UZ02_Freq_PV : ARRAY[0..0] OF WORD  // UZ_FREQUENCY_PV
            input  Application.GVL.UZ02_Status_Word : ARRAY[0..0] OF WORD  // UZ_STATUS
            output Application.GVL.UZ02_Freq_SP : ARRAY[0..0] OF WORD  // UZ_FREQUENCY_SP
            unmapped channels: UZ_CONTROL
        UZ01 : Modbus Slave, COM Port, 3S - Smart Software Solutions GmbH, version 3.5.10.30
            settings: SlaveAddress = 1; ResponseTimeout = 1000; UseExtendedFunctionCodes = TRUE; UZ_FREQUENCY_PV.Function Code = 3; UZ_FREQUENCY_PV.Read Offset = 16#C421; UZ_FREQUENCY_PV.Read Length = 1; UZ_FREQUENCY_PV.Write Offset = 0; UZ_FREQUENCY_PV.Write Length = 0; UZ_FREQUENCY_PV.Cycle Time = 100; UZ_STATUS.Function Code = 3; UZ_STATUS.Read Offset = 16#C417; UZ_STATUS.Read Length = 1; UZ_STATUS.Write Offset = 0; UZ_STATUS.Write Length = 0; UZ_STATUS.Cycle Time = 100; UZ_CONTROL.Function Code = 6; UZ_CONTROL.Read Offset = 0; UZ_CONTROL.Read Length = 0; UZ_CONTROL.Write Offset = 16#C34F; UZ_CONTROL.Write Length = 1; UZ_CONTROL.Cycle Time = 100; UZ_FREQUENCY_SP.Function Code = 6; UZ_FREQUENCY_SP.Read Offset = 0; UZ_FREQUENCY_SP.Read Length = 0; UZ_FREQUENCY_SP.Write Offset = 16#C359; UZ_FREQUENCY_SP.Write Length = 1; UZ_FREQUENCY_SP.Cycle Time = 100
            input  Application.GVL.UZ01_Freq_PV : ARRAY[0..0] OF WORD  // UZ_FREQUENCY_PV
            input  Application.GVL.UZ01_Status_Word : ARRAY[0..0] OF WORD  // UZ_STATUS
            output Application.GVL.UZ01_Freq_SP : ARRAY[0..0] OF WORD  // UZ_FREQUENCY_SP
            unmapped channels: UZ_CONTROL
        UZ14 : Modbus Slave, COM Port, 3S - Smart Software Solutions GmbH, version 3.5.10.30
            settings: SlaveAddress = 14; ResponseTimeout = 1000; UseExtendedFunctionCodes = TRUE; UZ_FREQUENCY_PV.Function Code = 3; UZ_FREQUENCY_PV.Read Offset = 16#C421; UZ_FREQUENCY_PV.Read Length = 1; UZ_FREQUENCY_PV.Write Offset = 0; UZ_FREQUENCY_PV.Write Length = 0; UZ_FREQUENCY_PV.Cycle Time = 100; UZ_STATUS.Function Code = 3; UZ_STATUS.Read Offset = 16#C417; UZ_STATUS.Read Length = 1; UZ_STATUS.Write Offset = 0; UZ_STATUS.Write Length = 0; UZ_STATUS.Cycle Time = 100; UZ_CONTROL.Function Code = 6; UZ_CONTROL.Read Offset = 0; UZ_CONTROL.Read Length = 0; UZ_CONTROL.Write Offset = 16#C34F; UZ_CONTROL.Write Length = 1; UZ_CONTROL.Cycle Time = 100; UZ_FREQUENCY_SP.Function Code = 6; UZ_FREQUENCY_SP.Read Offset = 0; UZ_FREQUENCY_SP.Read Length = 0; UZ_FREQUENCY_SP.Write Offset = 16#C359; UZ_FREQUENCY_SP.Write Length = 1; UZ_FREQUENCY_SP.Cycle Time = 100
            input  Application.GVL.UZ14_Freq_PV : ARRAY[0..0] OF WORD  // UZ_FREQUENCY_PV
            output Application.GVL.UZ14_Freq_SP : ARRAY[0..0] OF WORD  // UZ_FREQUENCY_SP
            unmapped channels: UZ_STATUS, UZ_CONTROL
    Screen : Screen, Production association OWEN, version 3.5.11.5002
        unmapped channels: Get Brightness, Dim time, Off time, Full brightness, Dim brightness, Off brightness, Dim visu name, Off visu name, On visu name, Wake up
    Network : Network, Production association OWEN, version 3.5.11.5002
        input  Application.TargetVars.stNetwork.xGetDhcp : BIT  // DHCP enabled
        input  Application.TargetVars.stNetwork.abyGetIp : ARRAY [0..3] OF BYTE  // IP
        input  Application.TargetVars.stNetwork.abyGetMask : ARRAY [0..3] OF BYTE  // Mask
        input  Application.TargetVars.stNetwork.abyGetGateway : ARRAY [0..3] OF BYTE  // Gateway
        input  Application.TargetVars.stNetwork.abyGetMac : ARRAY [0..5] OF BYTE  // MAC
        input  Application.TargetVars.stNetwork.sGetHostname : ARRAY [0..80] OF BYTE  // Hostname
        output Application.TargetVars.stNetwork.xSetDhcp : BIT  // Enable DHCP
        output Application.TargetVars.stNetwork.abySetIp : ARRAY [0..3] OF BYTE  // New IP
        output Application.TargetVars.stNetwork.abySetMask : ARRAY [0..3] OF BYTE  // New Mask
        output Application.TargetVars.stNetwork.abySetGateway : ARRAY [0..3] OF BYTE  // New Gateway
        output Application.TargetVars.stNetwork.sSetHostname : ARRAY [0..80] OF BYTE  // New Hostname
        output Application.TargetVars.stNetwork.xSetSettings : BIT  // Set Settings
    Buzzer : Buzzer, Production association OWEN, version 3.5.11.5002
        input  Application.TargetVars.stBuzzer.xGet : BIT  // Buzzer enabled
        output Application.TargetVars.stBuzzer.xSet : BIT  // Enable Buzzer
    OwenCloud : OwenCloud, Production association OWEN, version 3.5.11.5003
        unmapped channels: OwenCloud enabled, Folder error, Symbol error, Enable OwenCloud
  libraries: VisuSymbols, 3.5.10.0 (System)
  5ce3da45-db07-42e7-a21c-a00fff4ed8f6|Ленин - для мнемосхем\2-огр. паллет вверху.png
  5ce3da45-db07-42e7-a21c-a00fff4ed8f6|C:\Users\Alex\Desktop\LRF\IMG\M03UZ03_ON.png
  5ce3da45-db07-42e7-a21c-a00fff4ed8f6|Ленин - для мнемосхем\2-Подложка.png
  5ce3da45-db07-42e7-a21c-a00fff4ed8f6|C:\Users\Alex\Desktop\LRF\IMG\SQ04.png
  5ce3da45-db07-42e7-a21c-a00fff4ed8f6|Ленин - для мнемосхем\RUN-тр-р угловой.png
  5ce3da45-db07-42e7-a21c-a00fff4ed8f6|C:\Users\Alex\Desktop\LRF\IMG\M12KM12_ON.png
  5ce3da45-db07-42e7-a21c-a00fff4ed8f6|C:\Users\Alex\Desktop\LRF\IMG\SQ01.png
  5ce3da45-db07-42e7-a21c-a00fff4ed8f6|Ленин - для мнемосхем\2-пресс разжат.png
  5ce3da45-db07-42e7-a21c-a00fff4ed8f6|C:\Users\Alex\Desktop\LRF\IMG\M14UZ14_ON.png
  5ce3da45-db07-42e7-a21c-a00fff4ed8f6|Ленин - для мнемосхем\RUN-тр-р резчиковый.png
  5ce3da45-db07-42e7-a21c-a00fff4ed8f6|C:\Users\Alex\Desktop\LRF\IMG\SQ11.png
  5ce3da45-db07-42e7-a21c-a00fff4ed8f6|C:\Users\Alex\Desktop\LRF\IMG\SQ5.png
  5ce3da45-db07-42e7-a21c-a00fff4ed8f6|G:\Ленин - для мнемосхем\Подложка.png
  5ce3da45-db07-42e7-a21c-a00fff4ed8f6|C:\Users\Alex\Desktop\LRF\IMG\M01UZ01_ON.png
  5ce3da45-db07-42e7-a21c-a00fff4ed8f6|Ленин - для мнемосхем\RUN-тр-р выгружной.png
  5ce3da45-db07-42e7-a21c-a00fff4ed8f6|Ленин - для мнемосхем\2-выгрузчик сжат.png
  5ce3da45-db07-42e7-a21c-a00fff4ed8f6|G:\Ленин - для мнемосхем\RUN-тр-р резчиковый.png
  5ce3da45-db07-42e7-a21c-a00fff4ed8f6|C:\Users\Alex\Desktop\LRF\IMG\SQ06.png
  5ce3da45-db07-42e7-a21c-a00fff4ed8f6|C:\Users\Alex\Desktop\LRF\IMG\M05UZ05_ON.png
  5ce3da45-db07-42e7-a21c-a00fff4ed8f6|C:\Users\Alex\Desktop\LRF\IMG\M07KM07_ON.png
  5ce3da45-db07-42e7-a21c-a00fff4ed8f6|C:\Users\Alex\Desktop\LRF\IMG\RUN-PRES.png
  5ce3da45-db07-42e7-a21c-a00fff4ed8f6|Ленин - для мнемосхем\RUN-тр-р палетный.png
  5ce3da45-db07-42e7-a21c-a00fff4ed8f6|G:\Ленин - для мнемосхем\RUN-бункер-дозатор.png
  5ce3da45-db07-42e7-a21c-a00fff4ed8f6|C:\Users\Alex\Desktop\LRF\IMG\SQ10.png
  5ce3da45-db07-42e7-a21c-a00fff4ed8f6|C:\Users\Alex\Desktop\LRF\IMG\SQ02.png
  5ce3da45-db07-42e7-a21c-a00fff4ed8f6|Ленин - для мнемосхем\RUN-ПРФ.png
  5ce3da45-db07-42e7-a21c-a00fff4ed8f6|C:\Users\Alex\Desktop\LRF\IMG\SQ8.png
  5ce3da45-db07-42e7-a21c-a00fff4ed8f6|G:\транспортер.png
  5ce3da45-db07-42e7-a21c-a00fff4ed8f6|Ленин - для мнемосхем\2-паллет на погрузке - наличие кирпича.png
  5ce3da45-db07-42e7-a21c-a00fff4ed8f6|C:\Users\Alex\Desktop\LRF\IMG\SQ05.png
  5ce3da45-db07-42e7-a21c-a00fff4ed8f6|Ленин - для мнемосхем\RUN-горизонт прикатные ролики.png
  5ce3da45-db07-42e7-a21c-a00fff4ed8f6|Ленин - для мнемосхем\2-ПРФ позиция.png
  5ce3da45-db07-42e7-a21c-a00fff4ed8f6|C:\Users\Alex\Desktop\LRF\IMG\M08KM08_ON.png
  5ce3da45-db07-42e7-a21c-a00fff4ed8f6|C:\Users\Alex\Desktop\LRF\IMG\M09UZ09_ON.png
  5ce3da45-db07-42e7-a21c-a00fff4ed8f6|C:\Users\Alex\Desktop\LRF\IMG\SQ07.png
  5ce3da45-db07-42e7-a21c-a00fff4ed8f6|Ленин - для мнемосхем\RUN-пресс.png
  5ce3da45-db07-42e7-a21c-a00fff4ed8f6|Ленин - для мнемосхем\RUN-пресс ВНИЗУ.png
  text list GlobalTextList
  5ce3da45-db07-42e7-a21c-a00fff4ed8f6|Ленин - для мнемосхем\RUN-тр-р подающий.png
  5ce3da45-db07-42e7-a21c-a00fff4ed8f6|Ленин - для мнемосхем\RUN-пресс ВВЕРХУ.png
  5ce3da45-db07-42e7-a21c-a00fff4ed8f6|Ленин - для мнемосхем\2-выгрузчик разжат.png
  5ce3da45-db07-42e7-a21c-a00fff4ed8f6|Ленин - для мнемосхем\2-огр. паллет внизу.png
  5ce3da45-db07-42e7-a21c-a00fff4ed8f6|C:\Users\Alex\Desktop\LRF\IMG\Main.png
  5ce3da45-db07-42e7-a21c-a00fff4ed8f6|Ленин - для мнемосхем\RUN-вертик прикатной ролик.png
  5ce3da45-db07-42e7-a21c-a00fff4ed8f6|C:\Users\Alex\Desktop\LRF\IMG\MV01KM00_ON.png
  5ce3da45-db07-42e7-a21c-a00fff4ed8f6|C:\Users\Alex\Desktop\LRF\IMG\SQ9.png
  5ce3da45-db07-42e7-a21c-a00fff4ed8f6|C:\Users\sun_a\OneDrive\Рабочий стол\Obzor.png
  5ce3da45-db07-42e7-a21c-a00fff4ed8f6|Ленин - для мнемосхем\2-паллет на погрузке.png
  5ce3da45-db07-42e7-a21c-a00fff4ed8f6|Ленин - для мнемосхем\2-пресс сжат.png
  5ce3da45-db07-42e7-a21c-a00fff4ed8f6|C:\Users\Alex\Desktop\LRF\IMG\PRF.png
  5ce3da45-db07-42e7-a21c-a00fff4ed8f6|C:\Users\Alex\Desktop\LRF\IMG\SQ4.png
  5ce3da45-db07-42e7-a21c-a00fff4ed8f6|Ленин - для мнемосхем\RUN-тр-р существующий.png
  5ce3da45-db07-42e7-a21c-a00fff4ed8f6|C:\Users\Alex\Desktop\LRF\IMG\M11KM11_ON.png
  5ce3da45-db07-42e7-a21c-a00fff4ed8f6|C:\Users\Alex\Desktop\LRF\IMG\M06UZ06_ON.png
  5ce3da45-db07-42e7-a21c-a00fff4ed8f6|Ленин - для мнемосхем\2-паллет на очереди.png
  5ce3da45-db07-42e7-a21c-a00fff4ed8f6|C:\Users\Alex\Desktop\LRF\IMG\M04KM04_ON.png
*)

// Device/Application/TargetVariables/TRG_Drives
TYPE TRG_Drives :
STRUCT
	xEnable:			BOOL;
	
	uliFsFullSize: 		ULINT;
	uliFsUsedSize: 		ULINT;
	uliFsFreeSize: 		ULINT;
	
	xUsbMounted:		BOOL;
	xUsbUnmount:		BOOL;
	xUsbUnmountDone:	BOOL;
	
	uliUsbFullSize: 	ULINT;
	uliUsbUsedSize: 	ULINT;
	uliUsbFreeSize: 	ULINT;
	
	xSdMounted:			BOOL;
	xSdUnmount:			BOOL;
	xSdUnmountDone:		BOOL;
	
	uliSdFullSize: 		ULINT;
	uliSdUsedSize: 		ULINT;
	uliSdFreeSize: 		ULINT;
END_STRUCT
END_TYPE

// Device/Application/TargetVariables/TRG_Buzzer
TYPE TRG_Buzzer :
STRUCT
	xGet: 		BOOL;
	xSet: 		BOOL;
END_STRUCT
END_TYPE

// Device/Application/TargetVariables/TRG_RTC
TYPE TRG_RTC :
STRUCT
	uiGetYear:			UINT;
	usiGetMonth:		USINT;
	usiGetDay:			USINT;
	usiGetHour:			USINT;
	usiGetMinute:		USINT;
	usiGetSecond:		USINT;
	usiGetDayOfWeek:	USINT;
	usiGetWeekOfYear:	USINT;
	sGetFormatDate:		STRING;
	sGetFormatTime:		STRING;
	siGetUtcOffset:		USINT;
	dtDateAndTime:		DT;
	
	
	uiSetYear:			UINT;
	usiSetMonth:		USINT;
	usiSetDay:			USINT;
	usiSetHour:			USINT;
	usiSetMinute:		USINT;
	usiSetSecond:		USINT;
	siSetUtcOffset:		USINT;
	xUpdateSettings:	BOOL;
	
	xEnableNtp:			BOOL;
	xIsNtpEnabled:		BOOL;
	sPreferNtpServer:	STRING;
	usiNtpErrorCode:	USINT;
	
	ltSystemTick:		LTIME;
END_STRUCT
END_TYPE

// Device/Application/TargetVariables/TRG_Network
TYPE TRG_Network :
STRUCT
	xGetDhcp: 			BOOL;
	abyGetIp: 			ARRAY [0..3] OF BYTE;
	abyGetMask: 		ARRAY [0..3] OF BYTE;
	abyGetGateway: 		ARRAY [0..3] OF BYTE;
	abyGetMac: 			ARRAY [0..5] OF BYTE;
	sGetHostname: 		STRING;
	xSetDhcp: 			BOOL;
	abySetIp: 			ARRAY [0..3] OF BYTE;
	abySetMask: 		ARRAY [0..3] OF BYTE;
	abySetGateway: 		ARRAY [0..3] OF BYTE;
	sSetHostname: 		STRING;
	
	xSetSettings: 		BOOL;
END_STRUCT
END_TYPE

// Device/Application/TargetVariables/TRG_Info
TYPE TRG_Info :
STRUCT
	sVendorName: 			STRING;
	sDeviceName: 			STRING;
	sSerialId: 				STRING;
	sRuntimeVersion:		STRING;
	sFirmwareVersion: 		STRING;
	sLinuxVersion: 			STRING;
	sNeedTargetVersion:		STRING;
	
	sProjectName:			STRING;
	sAuthorName:			STRING;
	sProjectVersion:		STRING;
	sProjectProfile:		STRING;
	dtProjectLastChanges:	DT;
END_STRUCT
END_TYPE

// Device/Application/TargetVariables/TRG_Watchdog
TYPE TRG_Watchdog :
STRUCT
	eHandlingType:						Watchdog.ExceptionHandling;
	udiLastExceptionCode:				UDINT;
	sLastExceptionText:					STRING;
	dtLastExceptionTime:				DT;
	xIsHardwareWatchdogReboot:			BOOL;
	xDoReboot:							BOOL;
	usiPowerRebootCount:				USINT;
	usiExceptionRebootCount:			USINT;
	usiCommandRebootCount:				USINT;
	usiHardwareWatchdogRebootCount:		USINT;
	xResetCounters:						BOOL;
END_STRUCT
END_TYPE

// Device/Application/TargetVariables/TRG_Debug
TYPE TRG_Debug :
STRUCT
	xEnable: 			BOOL;
	udiPollingTime:		UDINT;
	udiRamUsedSize:		UDINT;
	udiRamFreeSize:		UDINT;
	udiCountHandles:	UDINT;
	udiProcUsage:		UDINT;
END_STRUCT
END_TYPE

// Device/Application/GVL
{attribute 'qualified_only'}
VAR_GLOBAL
//Преобразователь частоты UZ01 - Эл-двигатель дозатора (M01)
UZ01_Freq_SP 					: WORD;
UZ01_Freq_PV 					: WORD;
UZ01_Status_Word 				: WORD;
UZ01_Command_Word 				: WORD;
UZ01_Control_Ready 				: BOOL;
UZ01_Unit_Ready 				: BOOL;
UZ01_Alm_Stop 					: BOOL;
UZ01_Eror 						: BOOL;
UZ01_Block_Stop 				: BOOL;
UZ01_Warning 					: BOOL;
UZ01_Auto_Mode 					: BOOL;
UZ01_Running 					: BOOL;
UZ01_Reset_Alarm 				: BOOL;

//Преобразователь частоты UZ02 - Резервный (M02)
UZ02_Freq_SP 					: WORD;
UZ02_Freq_PV 					: WORD;
UZ02_Status_Word 				: WORD;
UZ02_Command_Word 				: WORD;
UZ02_Control_Ready 				: BOOL;
UZ02_Unit_Ready 				: BOOL;
UZ02_Alm_Stop 					: BOOL;
UZ02_Eror 						: BOOL;
UZ02_Block_Stop 				: BOOL;
UZ02_Warning 					: BOOL;
UZ02_Auto_Mode 					: BOOL;
UZ02_Running 					: BOOL;
UZ02_Reset_Alarm 				: BOOL;

//Преобразователь частоты UZ03 - Транспортер №1 (M03)
UZ03_Freq_SP 					: WORD;
UZ03_Freq_PV 					: WORD;
UZ03_Status_Word 				: WORD;
UZ03_Command_Word 				: WORD;
UZ03_Control_Ready 				: BOOL;
UZ03_Unit_Ready 				: BOOL;
UZ03_Alm_Stop 					: BOOL;
UZ03_Eror 						: BOOL;
UZ03_Block_Stop 				: BOOL;
UZ03_Warning 					: BOOL;
UZ03_Auto_Mode 					: BOOL;
UZ03_Running 					: BOOL;
UZ03_Reset_Alarm 				: BOOL;

//Преобразователь частоты UZ05 - Транспортер №2 (M05)
UZ05_Freq_SP 					: WORD;
UZ05_Freq_PV 					: WORD;
UZ05_Status_Word 				: WORD;
UZ05_Command_Word 				: WORD;
UZ05_Control_Ready 				: BOOL;
UZ05_Unit_Ready 				: BOOL;
UZ05_Alm_Stop 					: BOOL;
UZ05_Eror 						: BOOL;
UZ05_Block_Stop 				: BOOL;
UZ05_Warning 					: BOOL;
UZ05_Auto_Mode 					: BOOL;
UZ05_Running 					: BOOL;
UZ05_Reset_Alarm 				: BOOL;

//Преобразователь частоты UZ06 - Транспортер №3 (M06)
UZ06_Freq_SP 					: WORD;
UZ06_Freq_PV 					: WORD;
UZ06_Status_Word 				: WORD;
UZ06_Command_Word 				: WORD;
UZ06_Control_Ready 				: BOOL;
UZ06_Unit_Ready 				: BOOL;
UZ06_Alm_Stop 					: BOOL;
UZ06_Eror 						: BOOL;
UZ06_Block_Stop 				: BOOL;
UZ06_Warning 					: BOOL;
UZ06_Auto_Mode 					: BOOL;
UZ06_Running 					: BOOL;
UZ06_Reset_Alarm 				: BOOL;

//Преобразователь частоты UZ09 - Транспортер №5 (M09)
UZ09_Freq_SP 					: WORD;
UZ09_Freq_PV 					: WORD;
UZ09_Status_Word 				: WORD;
UZ09_Command_Word 				: WORD;
UZ09_Control_Ready 				: BOOL;
UZ09_Unit_Ready 				: BOOL;
UZ09_Alm_Stop 					: BOOL;
UZ09_Eror 						: BOOL;
UZ09_Block_Stop 				: BOOL;
UZ09_Warning 					: BOOL;
UZ09_Auto_Mode 					: BOOL;
UZ09_Running 					: BOOL;
UZ09_Reset_Alarm 				: BOOL;

//Преобразователь частоты UZ14 - Транспортер №8 (M14)
UZ14_Freq_SP 					: WORD;
UZ14_Freq_PV 					: WORD;
UZ14_Status_Word 				: WORD;
UZ14_Command_Word 				: WORD;
UZ14_Control_Ready 				: BOOL;
UZ14_Unit_Ready 				: BOOL;
UZ14_Alm_Stop 					: BOOL;
UZ14_Eror 						: BOOL;
UZ14_Block_Stop 				: BOOL;
UZ14_Warning 					: BOOL;
UZ14_Auto_Mode 					: BOOL;
UZ14_Running 					: BOOL;
UZ14_Reset_Alarm 				: BOOL;

//Преобразователь частоты UZ08 - Кантователь (M08)
UZ07_Freq_SP 					: WORD;
UZ07_Freq_PV 					: WORD;
UZ07_Status_Word 				: WORD;
UZ07_Command_Word 				: WORD;
UZ07_Control_Ready 				: BOOL;
UZ07_Unit_Ready 				: BOOL;
UZ07_Alm_Stop 					: BOOL;
UZ07_Block_Stop 				: BOOL;
UZ07_Eror 						: BOOL;
UZ07_Warning 					: BOOL;
UZ07_Auto_Mode 					: BOOL;
UZ07_Running 					: BOOL;
UZ07_Reset_Alarm 				: BOOL;

//Модуль дискретного ввода A1
A1_DI_Modul_Fail 				: BOOL;

A1_DI_QF25OK 					: BOOL;
A1_DI_QF26OK 					: BOOL;
A1_DI_380OK 					: BOOL;
A1_DI_SB_ALARM_STOP 			: BOOL;
A1_DI_SB_STOP 					: BOOL;
A1_DI_SB_1st_OPER 				: BOOL;  //SB21
A1_DI_SB_2nd_OPER 				: BOOL;  //SB35
A1_DI_SB_RESET 					: BOOL;
A1_DI_SB_START 					: BOOL;
A1_DI_SA01 						: BOOL;
// Кнопка "Тест"
	A1_DI_SB_TEST 					: BOOL;
A1_DI_MV01KM00_ON 				: BOOL;
A1_DI_M01UZ01_ON	 			: BOOL;
A1_DI_RESERV01		 			: BOOL;
A1_DI_M03UZ03_ON 				: BOOL;
A1_DI_M04KM04_ON 				: BOOL;
A1_DI_M05UZ05_ON 				: BOOL;
A1_DI_M06UZ06_ON 				: BOOL;
//Сост. "В РАБОТЕ" ПФР кантователь
A1_DI_M07KM07_ON 				: BOOL;
A1_DI_M08KM08_ON 				: BOOL;

//Модуль дискретного ввода A2
A2_DI_Modul_Fail 				: BOOL;

A2_DI_M09UZ09_ON 				: BOOL;
A2_DI_M10KM10_ON 				: BOOL;
A2_DI_M11KM11_ON 				: BOOL;
A2_DI_M12KM12_ON 				: BOOL;
A2_DI_M13KM13_ON 				: BOOL;
A2_DI_M14UZ14_ON 				: BOOL;
A2_DI_SQ01 						: BOOL;
A2_DI_SQ02						: BOOL;
A2_DI_SQ02_CLON 				: BOOL;
A2_DI_SQ02_CNT 					: UDINT;
// Останов резчика
	RESET_SQ2_CNT 					: BOOL;
// Запуск резчика
	A2_DI_SQ15 					: BOOL;
//Кирпич в конце
A2_DI_SQ03 						: BOOL;
A2_DI_RESERV02 					: BOOL;
//ПРФ, допресовщик разжат (исходное)
A2_DI_SQ04 						: BOOL;
//ПРФ, допресовщик сжат
A2_DI_SQ05 						: BOOL;
//ПРФ, выгрузчик разжат (исходное)
A2_DI_SQ06 						: BOOL;
//ПРФ, выгрузчик сжат (выталкивание)
A2_DI_SQ07 						: BOOL;
//ПРФ, позиционирование кантователя
A2_DI_SQ08 						: BOOL;
A2_DI_RESERV03 					: BOOL;
A2_DI_RESERV04 					: BOOL;
A2_DI_RESERV05 					: BOOL;
A2_DI_SQ09 						: BOOL;
A2_DI_SQ08_CLON 				: BOOL;
A2_DI_SQ08_CNT 					: UDINT;
RESET_CNT 						: BOOL;
//Модуль дискретного ввода A3
A3_DI_Modul_Fail 				: BOOL;

//Палет в зоне погрузки
A3_DI_SQ10 						: BOOL;
A3_DI_SQ13 						: BOOL;
A3_DI_SQ14 						: BOOL;
A3_DI_RESERV01 					: BOOL;
//Наличие кирпича на палете 
A3_DI_SQ11 						: BOOL;
A3_DI_SQ12 						: BOOL;
A3_DI_RESERV02 					: BOOL;
A3_DI_KV301 					: BOOL;
A3_DI_KV302 					: BOOL;
A3_DI_PI01 						: BOOL;
A3_DI_RESERV03 					: BOOL;
A3_DI_RESERV04 					: BOOL;
A3_DO_KV303 					: BOOL;
A3_DO_KV304 					: BOOL;
A3_DO_RESERV01 					: BOOL;
A3_DO_RESERV02 					: BOOL;

//Модуль дискретного ввода A4
A4_DI_Modul_Fail 				: BOOL;

A4_DO_HL02_32 					: BOOL;
A4_DO_HL21 						: BOOL;
A4_DO_HL35 						: BOOL;
A4_DO_HL03_33 					: BOOL;
A4_DO_HL04_34 					: BOOL;
A4_DO_HL05 						: BOOL;
A4_DO_XV01KV207 				: BOOL;
A4_DO_XV02KV208 				: BOOL;
A4_DO_XV03KV209 				: BOOL;
// Выход Малая скорость Кантователя (A4 вых.10->KV210->KM8
	A4_DO_XV04KV210 				: BOOL;
A4_DO_XV05KV211 				: BOOL;
A4_DO_XV06KV212 				: BOOL;
A4_DO_RESERV01 					: BOOL;
A4_DO_RESERV02 					: BOOL;
A5_DO_M02UZ02_RUN_REV 			: BOOL;
A4_DO_RESERV04 					: BOOL;

//Модуль дискретного ввода A5
A5_DI_Modul_Fail 				: BOOL;

A5_DO_MV01KM00_RUN 				: BOOL;
A5_DO_M01UZ01_RUN 				: BOOL;
A5_DO_M02UZ02_RUN_FORW 			: BOOL;
A5_DO_M03UZ03_RUN 				: BOOL;
A5_DO_M04KM04_RUN 				: BOOL;
A5_DO_M05UZ05_RUN 				: BOOL;
A5_DO_M06UZ06_RUN 				: BOOL;
// Выход Работа/Тормоз Кантователя (A5 вых.8  KV224->КM7)
	A5_DO_M07KM07_RUN 				: BOOL;
A5_DO_M08KM08_RUN 				: BOOL;
A5_DO_M09UZ09_RUN 				: BOOL;
// Двигатель маслостанции
	A5_DO_M10KM10_RUN 				: BOOL;
A5_DO_M11KM11_RUN 				: BOOL;
A5_DO_M12KM12_RUN 				: BOOL;
A5_DO_M13KM13_RUN 				: BOOL;
A5_DO_M14UZ14_RUN 				: BOOL;
A5_DO_RESERV01 					: BOOL;

//Дата и время для HMI
PLC_DATE 						: STRING[80];
PLC_TIME 						: STRING[80];

(*Состояния ЛРФ*)
LRF_MODE 						: INT;
LRF_AUTO 						: BOOL;
// ЛРФ в режиме "ТЕСТ"
	LRF_TEST 						: BOOL;
LRF_MANUAL 						: BOOL;

LRFRDYSTS						: BOOL;
LRFRUNSTS 						: BOOL;

(*Аварии*)
LRFALMSTS 						: BOOL;
ALMACK 							: BOOL;

A1_DI_QF25OK_ALM 				: BOOL;
A1_DI_QF26OK_ALM 				: BOOL;
A1_DI_380OK_ALM 				: BOOL; 
A2_DI_SQ06_ALM 					: BOOL;

XV01KV207_ALM 					: BOOL;
XV02KV208_ALM 					: BOOL;
XV03KV209_ALM 					: BOOL;
XV04KV210_ALM 					: BOOL;
XV05KV211_ALM 					: BOOL;
XV06KV212_ALM 					: BOOL;
MV01KM00_ALM 					: BOOL;
M01UZ01_ALM 					: BOOL;
M02UZ02_ALM						: BOOL;
M03UZ03_ALM 					: BOOL;
M04KM04_ALM 					: BOOL;
M05UZ05_ALM 					: BOOL;
M06UZ06_ALM 					: BOOL;
M07KM07_ALM						: BOOL;
M08KM08_ALM 					: BOOL;
M09UZ09_ALM						: BOOL;
M10KM10_ALM						: BOOL;
M11KM11_ALM						: BOOL;
M12KM12_ALM						: BOOL;
M13KM13_ALM						: BOOL;
M14UZ14_ALM						: BOOL;
PI01_ALM 						: BOOL;
SQ08_ALM 						: BOOL;


(*Управление ИМ*)
TSTOI 							: INT;
XV01KV207_TSTOI 				: BOOL;
XV02KV208_TSTOI 				: BOOL;
XV03KV209_TSTOI 				: BOOL;
XV04KV210_TSTOI 				: BOOL;
XV05KV211_TSTOI 				: BOOL;
XV06KV212_TSTOI 				: BOOL;
MV01KM00_TSTOI 					: BOOL;
M01UZ01_TSTOI 					: BOOL;
M02UZ02_TSTOI					: BOOL;
M03UZ03_TSTOI 					: BOOL;
M04KM04_TSTOI 					: BOOL;
M05UZ05_TSTOI 					: BOOL;
M06UZ06_TSTOI 					: BOOL;
M07KM07_TSTOI					: BOOL;
M08KM08_TSTOI 					: BOOL;
M09UZ09_TSTOI					: BOOL;
M10KM10_TSTOI					: BOOL;
M11KM11_TSTOI					: BOOL;
M12KM12_TSTOI					: BOOL;
M13KM13_TSTOI					: BOOL;
M14UZ14_TSTOI					: BOOL;

(*Управление ИМ*)
CFGOI 							: INT;
XV01KV207_CFGOI 				: BOOL;
XV02KV208_CFGOI 				: BOOL;
XV03KV209_CFGOI 				: BOOL;
XV04KV210_CFGOI 				: BOOL;
XV05KV211_CFGOI 				: BOOL;
XV06KV212_CFGOI 				: BOOL;
MV01KM00_CFGOI 					: BOOL;
// Задействовать
	M01UZ01_CFGOI 					: BOOL := FALSE;
M02UZ02_CFGOI					: BOOL;
M03UZ03_CFGOI 					: BOOL := TRUE;
M04KM04_CFGOI 					: BOOL;
M05UZ05_CFGOI 					: BOOL := TRUE;
M06UZ06_CFGOI 					: BOOL := TRUE;
M07KM07_CFGOI					: BOOL;
M08KM08_CFGOI 					: BOOL;
M09UZ09_CFGOI					: BOOL;
M10KM10_CFGOI					: BOOL;
M11KM11_CFGOI					: BOOL := TRUE;
M12KM12_CFGOI					: BOOL := TRUE;
M13KM13_CFGOI					: BOOL;
M14UZ14_CFGOI					: BOOL := TRUE;

XV01KV207_MANOI 				: BOOL;
XV02KV208_MANOI 				: BOOL;
XV03KV209_MANOI 				: BOOL;
XV04KV210_MANOI 				: BOOL;
XV05KV211_MANOI 				: BOOL;
XV06KV212_MANOI 				: BOOL;
MV01KM00_MANOI 					: BOOL;
M01UZ01_MANOI 					: BOOL;
M02UZ02_MANOI					: BOOL;
M03UZ03_MANOI 					: BOOL;
M04KM04_MANOI 					: BOOL;
M05UZ05_MANOI 					: BOOL;
M06UZ06_MANOI 					: BOOL;
// Работа/Тормоз Кантователя Ручной
	M07KM07_MANOI					: BOOL;
M08KM08_MANOI 					: BOOL;
M09UZ09_MANOI					: BOOL;
M10KM10_MANOI					: BOOL;
M11KM11_MANOI					: BOOL;
M12KM12_MANOI					: BOOL;
M13KM13_MANOI					: BOOL;
M14UZ14_MANOI					: BOOL;

XV01KV207_AUX 					: BOOL;
XV02KV208_AUX 					: BOOL; (*команда разжатие формы*)
XV03KV209_AUX 					: BOOL;
XV04KV210_AUX 					: BOOL;
XV05KV211_AUX 					: BOOL;
XV06KV212_AUX 					: BOOL;
MV01KM00_AUX 					: BOOL;
M01UZ01_AUX 					: BOOL;
M02UZ02_AUX						: BOOL;
M03UZ03_AUX 					: BOOL;
M04KM04_AUX 					: BOOL;
M05UZ05_AUX 					: BOOL;
M06UZ06_AUX 					: BOOL;
M07KM07_AUX						: BOOL;
M08KM08_AUX 					: BOOL;
M09UZ09_AUX						: BOOL;
M10KM10_AUX						: BOOL;
M11KM11_AUX						: BOOL;
M12KM12_AUX						: BOOL;
M13KM13_AUX						: BOOL;
M14UZ14_AUX						: BOOL;

(*Фактическая частота*)
M01UZ01_PV 						: INT;
M02UZ02_PV						: INT;
M03UZ03_PV 						: INT;
M05UZ05_PV 						: INT;
M06UZ06_PV 						: INT;
M09UZ07_PV						: INT;
M09UZ09_PV						: INT;
M14UZ14_PV						: INT;

A1_DI_SB_1st_OPER_KEEP 			:BOOL;
A1_DI_SB_2nd_OPER_KEEP 			:BOOL;










END_VAR

// Device/Application/TargetVariables/TargetVars
{attribute 'qualified_only'}
VAR_GLOBAL
	stBuzzer:	 TRG_Buzzer;
	stDebug: 	 TRG_Debug;
	stDrives: 	 TRG_Drives;
	stNetwork:	 TRG_Network;
	stRtc:		 TRG_RTC;
	stInfo:		 TRG_Info;
	stWatchdog:	 TRG_Watchdog;
END_VAR

// Device/Application/GVLR
{attribute 'qualified_only'}
VAR_GLOBAL RETAIN
(*Таймера задержки запуска*)	
TIME_XV01KV207_DELAY 			: INT;
TIME_XV02KV208_DELAY 			: INT;
TIME_XV03KV209_DELAY 			: INT;
// Время отключения выталкивателя (S)
	TIME_XV03KV209_UP 				: INT := 3;
TIME_XV04KV210_DELAY 			: INT;
TIME_XV05KV211_DELAY 			: INT;
TIME_XV06KV212_DELAY 			: INT;
TIME_MV01KM00_ON	 			: INT;
TIME_MV01KM00_OFF	 			: INT;
TIME_M01UZ01_DELAY 				: INT;
TIME_M02UZ02_DELAY				: INT;
TIME_M03UZ03_DELAY 				: INT;
TIME_M04KM04_DELAY 				: INT;
TIME_M05UZ05_DELAY 				: INT;
TIME_M06UZ06_DELAY 				: INT;
	// Задержка включения малой скорости
	TIME_SPEED2_DELAY: REAL := 2.15;
TIME_M07KM07_DELAY				: INT;
TIME_M08KM08_DELAY 				: INT;
TIME_M08KM08_OFF 				: INT;
TIME_M09UZ09_DELAY				: INT;
TIME_M09UZ09_OFF				: INT := 11;
TIME_M10KM10_DELAY				: INT;
TIME_M11KM11_DELAY				: INT;
TIME_M12KM12_DELAY				: INT;
TIME_M13KM13_DELAY				: INT;
TIME_M14UZ14_DELAY				: INT;
TIME_M14UZ14_OFF				: INT;

(*Аварийные таймера*)
TIME_XV01KV207_ALM 				: INT := 5;
TIME_XV02KV208_ALM 				: INT := 5;
TIME_XV03KV209_ALM 				: INT := 5;
TIME_XV04KV210_ALM 				: INT := 5;
TIME_XV05KV211_ALM 				: INT := 5;
TIME_XV06KV212_ALM 				: INT := 5;
TIME_MV01KM00_ALM 				: INT := 5;
TIME_M01UZ01_ALM 				: INT := 5;
TIME_M02UZ02_ALM				: INT := 5;
TIME_M03UZ03_ALM 				: INT := 5;
TIME_M04KM04_ALM 				: INT := 5;
TIME_M05UZ05_ALM 				: INT := 5;
TIME_M06UZ06_ALM 				: INT := 5;
TIME_M07KM07_ALM				: INT := 5;
TIME_M08KM08_ALM 				: INT := 5;
TIME_M09UZ09_ALM				: INT := 5;
TIME_M10KM10_ALM				: INT := 5;
TIME_M11KM11_ALM				: INT := 5;
TIME_M12KM12_ALM				: INT := 5;
TIME_M13KM13_ALM				: INT := 5;
TIME_M14UZ14_ALM				: INT := 5;
TIME_PI01_ALM 					: INT := 10;
TIME_SQ08_ALM 					: INT := 10;
TIME_SQ06_ALM 					: INT := 10;

(*Задания для частотников*)
M01UZ01_SP 						: WORD := 10;
M02UZ02_SP						: WORD := 20;
M03UZ03_SP 						: WORD := 50;
M05UZ05_SP 						: WORD := 50;
M06UZ06_SP 						: WORD := 50;
M09UZ07_SP1						: WORD;
M09UZ07_SP2						: WORD;
M09UZ09_SP						: WORD := 25;
M14UZ14_SP						: WORD := 20;

(*Sequencer*)
PRF_STEPS 						: INT;
PRF_STEP1						: BOOL;
PRF_STEP2 						: BOOL;
PRF_STEP3 						: BOOL;
PRF_STEP4 						: BOOL;
PRF_STEP5 						: BOOL;
PRF_STEP6 						: BOOL;
PRF_STEP_DONE 					: BOOL;
PRF_SHIFT_STEP 					: BOOL;
	// Счетчик Циклов ПФР
	PRF_COUNTER_AUTO: DWORD;
	TIMER_SQ5_DELAY: REAL := 0.5;
END_VAR

// Device/Application/Main
PROGRAM Main
VAR
	ONE_SEC_IMP 				: BOOL;
	IMP 						: BLINK;
	A1_DI_SB_START_OSR 			: R_TRIG;
	A1_DI_SB_STOP_OSR 			: R_TRIG;
	LAMPTEST 					: BOOL;
	LAMPTEST_TIM 				: TON;
	A1_DI_SB_1st_OPER_OSR 		: R_TRIG;
	A1_DI_SB_2nd_OPER_OSR		: R_TRIG;
	A1_DI_SB_1st_OPER_KEEP 		: BOOL;
	A1_DI_SB_2nd_OPER_KEEP 		: BOOL;
	SP 							: WORD;
	SET_SETTINGS 				: BOOL;
	
END_VAR

(*Импульс 1 сек*)
IMP(ENABLE:= TRUE, TIMELOW:= T#1S, TIMEHIGH:= T#1S, OUT=> ONE_SEC_IMP);

(*Режим управления ЛРФ*)
GVL.LRF_AUTO := GVL.LRF_MODE = 1;
GVL.LRF_TEST := GVL.LRF_MODE = 2;
GVL.LRF_MANUAL := GVL.LRF_MODE = 3;
(**)
IF NOT GVL.A1_DI_SA01 THEN
	GVL.LRF_MODE := 0;
END_IF;


(*Кнопки управления*)
A1_DI_SB_START_OSR(CLK:= GVL.A1_DI_SB_START);
A1_DI_SB_STOP_OSR(CLK:= GVL.A1_DI_SB_STOP);
A1_DI_SB_1st_OPER_OSR(CLK:= GVL.A1_DI_SB_1st_OPER);
A1_DI_SB_2nd_OPER_OSR(CLK:= GVL.A1_DI_SB_2nd_OPER);

GVL.LRFRDYSTS := GVL.LRF_MODE > 0 AND NOT GVL.LRFALMSTS AND GVL.A1_DI_SA01;
(**)
IF A1_DI_SB_START_OSR.Q AND GVL.LRFRDYSTS AND GVL.LRF_AUTO THEN
	GVL.LRFRUNSTS := TRUE;
	ELSIF NOT GVL.LRF_AUTO OR NOT GVL.LRFRDYSTS OR A1_DI_SB_STOP_OSR.Q THEN
		GVL.LRFRUNSTS := FALSE;
END_IF;

GVL.A3_DO_KV303 := GVL.LRFRUNSTS AND GVL.A1_DI_M03UZ03_ON;

(*Индикаторные лампы на шкафу управления*)
LAMPTEST_TIM(IN:= GVL.A1_DI_SB_RESET, PT:= T#3S);
LAMPTEST := LAMPTEST_TIM.Q;
GVL.A4_DO_HL04_34 := (GVL.LRF_AUTO AND GVL.LRFRDYSTS AND NOT GVL.LRFRUNSTS AND ONE_SEC_IMP) OR GVL.LRFRUNSTS OR LAMPTEST;

GVL.A4_DO_HL02_32 := (NOT GVL.LRFRUNSTS AND GVL.LRFRDYSTS AND NOT GVL.LRFALMSTS AND GVL.A1_DI_SA01) OR
					  LAMPTEST;
					  
GVL.A4_DO_HL05 := (GVL.LRF_TEST AND GVL.LRFRDYSTS AND NOT GVL.LRFALMSTS) OR LAMPTEST;

GVL.A4_DO_HL03_33 := (GVL.LRFALMSTS AND ONE_SEC_IMP) OR LAMPTEST;

GVL.A4_DO_HL21 := (GVL.LRF_AUTO AND NOT A1_DI_SB_1st_OPER_KEEP AND ONE_SEC_IMP AND GVL.LRFRUNSTS) OR (GVL.A1_DI_SB_1st_OPER_KEEP AND GVL.LRF_AUTO) OR LAMPTEST;

GVL.A4_DO_HL35 := (GVL.LRF_AUTO AND NOT A1_DI_SB_2nd_OPER_KEEP AND ONE_SEC_IMP AND GVL.LRFRUNSTS) OR (GVL.A1_DI_SB_2nd_OPER_KEEP AND GVL.LRF_AUTO) OR LAMPTEST;

(*Тестовый режим*)
GVL.XV01KV207_TSTOI 	:= GVL.TSTOI = 1;
GVL.XV02KV208_TSTOI 	:= GVL.TSTOI = 2;
GVL.XV03KV209_TSTOI 	:= GVL.TSTOI = 3;
GVL.XV04KV210_TSTOI 	:= GVL.TSTOI = 4;
GVL.MV01KM00_TSTOI 		:= GVL.TSTOI = 5;
GVL.M01UZ01_TSTOI 		:= GVL.TSTOI = 6;
GVL.M03UZ03_TSTOI 		:= GVL.TSTOI = 7;
GVL.M02UZ02_TSTOI 		:= GVL.TSTOI = 8;
GVL.M05UZ05_TSTOI 		:= GVL.TSTOI = 9;
GVL.M06UZ06_TSTOI 		:= GVL.TSTOI = 10;
GVL.M07KM07_TSTOI 		:= GVL.TSTOI = 11; (*Выбор Кантователя*)
GVL.M08KM08_TSTOI 		:= GVL.TSTOI = 12;
GVL.M09UZ09_TSTOI 		:= GVL.TSTOI = 13;
GVL.M10KM10_TSTOI 		:= GVL.TSTOI = 14;
GVL.M11KM11_TSTOI 		:= GVL.TSTOI = 15;
GVL.M12KM12_TSTOI 		:= GVL.TSTOI = 16;
GVL.M14UZ14_TSTOI 		:= GVL.TSTOI = 17;

IF NOT GVL.LRF_TEST THEN
	GVL.TSTOI := 0;
END_IF;

(*Автомат кантователя*)

IF GVL.LRF_AUTO AND A1_DI_SB_1st_OPER_OSR.Q AND GVL.LRFRUNSTS (*AND NOT GVL.A3_DI_SQ11 AND GVL.A3_DI_SQ10*) THEN
	GVL.A1_DI_SB_1st_OPER_KEEP := TRUE;
END_IF;

IF GVL.LRF_AUTO AND A1_DI_SB_2nd_OPER_OSR.Q AND GVL.LRFRUNSTS (*AND NOT GVL.A3_DI_SQ11 AND GVL.A3_DI_SQ10*)  THEN
	GVL.A1_DI_SB_2nd_OPER_KEEP := TRUE;
END_IF;

GVL.UZ01_Freq_SP := GVLR.M01UZ01_SP * 328;
GVL.UZ02_Freq_SP := GVLR.M02UZ02_SP * 328;
GVL.UZ03_Freq_SP := GVLR.M03UZ03_SP * 328; 
GVL.UZ05_Freq_SP := GVLR.M05UZ05_SP * 328;
GVL.UZ06_Freq_SP := GVLR.M06UZ06_SP * 328;
GVL.UZ09_Freq_SP := GVLR.M09UZ09_SP * 328;
GVL.UZ14_Freq_SP := GVLR.M14UZ14_SP * 328;

IF SET_SETTINGS THEN
GVLR.TIME_XV01KV207_ALM := 10;
GVLR.TIME_XV02KV208_ALM := 20;
GVLR.TIME_XV03KV209_ALM := 10;
GVLR.TIME_XV04KV210_ALM := 10;
GVLR.TIME_XV05KV211_ALM := 10;
GVLR.TIME_XV06KV212_ALM := 10;
GVLR.TIME_MV01KM00_ALM := 10;
GVLR.TIME_M01UZ01_ALM := 10;
GVLR.TIME_M02UZ02_ALM := 10;
GVLR.TIME_M03UZ03_ALM := 10;
GVLR.TIME_M04KM04_ALM := 10;
GVLR.TIME_M05UZ05_ALM := 10;
GVLR.TIME_M06UZ06_ALM := 10;
GVLR.TIME_M07KM07_ALM := 20;
GVLR.TIME_M08KM08_ALM := 10;
GVLR.TIME_M09UZ09_ALM := 10;
GVLR.TIME_M10KM10_ALM := 10;
GVLR.TIME_M11KM11_ALM := 10;
GVLR.TIME_M12KM12_ALM := 10;
GVLR.TIME_M13KM13_ALM := 10;
GVLR.TIME_M14UZ14_ALM := 10;
GVLR.TIME_PI01_ALM := 90;
GVLR.TIME_SQ08_ALM := 50;
GVLR.TIME_SQ06_ALM := 11;	
END_IF;

END_PROGRAM

// Device/Application/Alarm
PROGRAM Alarm
VAR

END_VAR

GVL.ALMACK := GVL.A1_DI_SB_RESET;

GVL.A1_DI_QF25OK_ALM := NOT GVL.A1_DI_QF25OK OR (GVL.A1_DI_QF25OK_ALM AND NOT GVL.ALMACK);
GVL.A1_DI_QF26OK_ALM := NOT GVL.A1_DI_QF26OK OR (GVL.A1_DI_QF26OK_ALM AND NOT GVL.ALMACK);
GVL.A1_DI_380OK_ALM := NOT GVL.A1_DI_380OK OR (GVL.A1_DI_380OK_ALM AND NOT GVL.ALMACK);

GVL.LRFALMSTS := NOT GVL.A1_DI_SB_ALARM_STOP OR GVL.A1_DI_QF25OK_ALM OR GVL.A1_DI_QF26OK_ALM OR
				 GVL.A1_DI_380OK_ALM OR GVL.XV01KV207_ALM OR GVL.XV02KV208_ALM OR GVL.XV03KV209_ALM OR 
				 GVL.XV04KV210_ALM OR GVL.MV01KM00_ALM OR GVL.M01UZ01_ALM OR GVL.M03UZ03_ALM OR GVL.M04KM04_ALM OR 
				 GVL.M05UZ05_ALM OR GVL.M06UZ06_ALM OR GVL.M07KM07_ALM OR GVL.M08KM08_ALM OR GVL.M09UZ09_ALM OR 
				 GVL.M10KM10_ALM OR GVL.M11KM11_ALM OR GVL.M12KM12_ALM OR GVL.M14UZ14_ALM OR GVL.PI01_ALM OR GVL.SQ08_ALM OR 
				 GVL.A2_DI_SQ06_ALM;

END_PROGRAM

// Device/Application/Motors
PROGRAM Motors
VAR
	(*Кантователь M07KM07*)
	M07KM07_ALM_TIM 		: TON;
	M07KM07_SUM 			: BOOL;
	M07KM07_AUX_TIM 		: TON;
	A2_DI_SQ08_OSR 			: R_TRIG;
	A2_DI_SQ08_KEEP 		: BOOL;
	SQ08_ALM_TIM 			: TON;
	M07KM07_RUN_TIM 		: TON;
	// Большая скорость кантователя
	SPEED1 					: BOOL;
	// Малая скорость кантователя
	SPEED2 					: BOOL;
	M07KM07_RUN_TIM_ET 		: TIME;
	SQ08_TIM 				: TON;
	SQ08_ON_TIM 			: TON;
	(*Пресс XV01KV207*)
	XV01KV207_ALM_TIM 		: TON;
	XV01KV207_SUM 			: BOOL;
	XV01KV207_AUX_TIM 		: TON;
	SQ05_TIM 				: TON;
	(*Пресс XV02KV208*)
	XV02KV208_ALM_TIM 		: TON;
	XV02KV208_SUM 			: BOOL;
	// Таймер разжатия формы
	XV02KV208_AUX_TIM 		: TON;
	XV03KV209_ALM_TIM 		: TON;
	XV03KV209_SUM 			: BOOL;
	XV03KV209_AUX_TIM 		: TON;
	XV03KV209_AUX_UP		: TON;
	SQ04_SR 				: SR;
	(*Маслостанция*)
	M10KM10_ALM_TIM 		: TON;
	M10KM10_SUM 			: BOOL;
	PI01_ALM_TIM 			: TON;
	(*Выталкиватель XV03KV209*)
	XV04KV210_ALM_TIM 		: TON;
	XV04KV210_SUM 			: BOOL;
	XV04KV210_AUX_TIM 		: TON;
	SQ06_SR 				: SR;
	SQ10_SR 			: SR;
	(*MV01KM00_RUN*)
	MV01KM00_SUM 			: BOOL;
	MV01KM00_AUX_TIM 		: TON;
	MV01KM00_ALM_TIM 		: TON;
	MV01KM00_ON_TIM 		: TON;
	MV01KM00_OFF_TIM 		: TON;
	MV01KM00_IMP 			: BLINK;
	(*M01UZ01_RUN*)
	M01UZ01_SUM 			: BOOL;
	M01UZ01_AUX_TIM 		: TON;
	M01UZ01_ALM_TIM 		: TON;
	M02UZ02_SUM 			: BOOL;
	M02UZ02_AUX_TIM 		: TON;
	M02UZ02_ALM_TIM 		: TON;
	M02UZ02_SR 				: SR;
	M02UZ02_START 			: BOOL;
	A2_DI_SQ15_OSR 			: R_TRIG;
	A2_DI_SQ02_OSR 			: R_TRIG;
	M03UZ03_SUM 			: BOOL;
	M03UZ03_AUX_TIM 		: TON;
	M03UZ03_ALM_TIM 		: TON;
	M05UZ05_SUM 			: BOOL;
	M05UZ05_AUX_TIM 		: TON;
	M05UZ05_ALM_TIM 		: TON;
	M06UZ06_SUM 			: BOOL;
	M06UZ06_AUX_TIM 		: TON;
	M06UZ06_ALM_TIM 		: TON;
	M08KM08_SUM 			: BOOL;
	M08KM08_AUX_TIM 		: TON;
	M08KM08_ALM_TIM 		: TON;
	M08KM08_SR 				: SR;
	M08KM08_AUX_OFF 		: TON;
	M09UZ09_SUM 			: BOOL;
	M09UZ09_AUX_TIM 		: TON;
	M09UZ09_AUX_OFF 		: TON;
	M09UZ09_SR 				: SR;
	M09UZ09_START 			: BOOL;
	M09UZ09_ALM_TIM 		: TON;
	M09UZ09_READY_TO_RUN    : BOOL;
	A2_DI_SQ06_ALM_TIM 		: TON;
	A3_DI_SQ11_TIM		 	: TON;
	M14UZ14_SUM 			: BOOL;
	M14UZ14_AUX_TIM 		: TON;
	M14UZ14_ALM_TIM 		: TON;
	M14UZ14_SR 				: SR;
	M14UZ14_AUX_OFF 		: TON;
	M11KM11_SUM 			: BOOL;
	M11KM11_AUX_TIM 		: TON;
	M11KM11_ALM_TIM 		: TON;
	M12KM12_SUM 			: BOOL;
	M12KM12_AUX_TIM 		: TON;
	M12KM12_ALM_TIM 		: TON;
	// Задержка запуска кантователя
	Delay_M07_Run: INT;
	T_SPEED2_DELAY: TIME;
	// Временное состояние SQ2
	TEMP_SQ2_CLON: BOOL;
	TON_SQ15: TON;
	SQ15_QSR: R_TRIG;
	M07KM07_R_TRIG: R_TRIG;
END_VAR

(*Кантователь M07KM07*)

GVL.RESET_CNT := NOT GVL.A5_DO_M07KM07_RUN;
GVL.M07KM07_ALM := M07KM07_ALM_TIM.Q OR (GVL.M07KM07_ALM AND NOT GVL.ALMACK);
(*
M07KM07_ALM_TIM(IN:= (GVL.A5_DO_M07KM07_RUN AND NOT GVL.A1_DI_M07KM07_ON) OR 
					 (NOT GVL.A5_DO_M07KM07_RUN AND GVL.A1_DI_M07KM07_ON),
				PT:= INT_TO_TIME(GVLR.TIME_M07KM07_ALM * 1000));*)
				
GVL.SQ08_ALM := SQ08_ALM_TIM.Q OR (GVL.SQ08_ALM AND NOT GVL.ALMACK);
SQ08_ALM_TIM(IN:= (GVL.A5_DO_M07KM07_RUN AND NOT GVL.A2_DI_SQ08),
			 PT:= INT_TO_TIME(GVLR.TIME_SQ08_ALM * 1000)); 

SQ06_SR(SET1:= NOT GVL.A4_DO_XV03KV209 AND GVL.A2_DI_SQ06, 
		RESET:= GVL.A4_DO_XV03KV209);

SQ04_SR(SET1:= NOT GVL.A4_DO_XV02KV208 AND GVL.A2_DI_SQ04, 
		RESET:= GVL.A4_DO_XV02KV208);
				
M07KM07_SUM := (*GVL.A2_DI_SQ06*) SQ06_SR.Q1 AND (*GVL.A2_DI_SQ04*) SQ04_SR.Q1 AND NOT GVL.A4_DO_XV03KV209 AND 
			   (*NOT GVL.A3_DI_SQ11 AND GVL.A3_DI_SQ10 AND *)GVL.LRFRDYSTS;

SQ08_TIM(IN:= (GVL.A1_DI_M07KM07_ON),
			   PT:= T#2S);

GVL.A2_DI_SQ08_CLON := GVL.A2_DI_SQ08_CNT > 0 AND SQ08_TIM.Q;

SQ08_ON_TIM(IN:= (GVL.A2_DI_SQ08_CLON AND GVL.A2_DI_SQ08),
			   PT:= T#0.1S);

A2_DI_SQ08_OSR(CLK:= SQ08_ON_TIM.Q (*GVL.A2_DI_SQ08_CLON*));
(**)
IF  GVL.LRF_AUTO AND GVL.LRFRUNSTS AND A2_DI_SQ08_OSR.Q (*AND GVL.A1_DI_M07KM07_ON*) THEN
	A2_DI_SQ08_KEEP := TRUE;
	(*ELSIF NOT GVL.A1_DI_M07KM07_ON THEN
		A2_DI_SQ08_KEEP := FALSE;*)
END_IF;

IF GVL.LRF_MANUAL AND (A2_DI_SQ08_OSR.Q AND GVL.A1_DI_M07KM07_ON) OR NOT M07KM07_SUM OR NOT GVL.LRF_MANUAL THEN
	GVL.M07KM07_MANOI := FALSE; (*Работа/Торможение кантователя*)
END_IF;

GVL.M07KM07_AUX := (GVL.LRF_TEST AND GVL.M07KM07_TSTOI AND M07KM07_SUM AND GVL.A1_DI_SB_TEST (*AND NOT A2_DI_SQ08_KEEP*)) OR
				   (*(GVL.LRF_MANUAL AND GVL.M07KM07_MANOI AND M07KM07_SUM AND NOT A2_DI_SQ08_KEEP) OR*)
				   (GVL.LRF_AUTO AND M07KM07_SUM AND NOT A2_DI_SQ08_KEEP AND (GVL.A1_DI_SB_1st_OPER_KEEP OR
					GVL.A1_DI_SB_2nd_OPER_KEEP) AND GVL.LRFRUNSTS);
					
T_SPEED2_DELAY := REAL_TO_TIME (GVLR.TIME_SPEED2_DELAY * 1000);
M07KM07_RUN_TIM(IN:= M07KM07_AUX_TIM.Q AND GVL.LRF_AUTO,
				PT:= T_SPEED2_DELAY); (*Задержка переключения на малую скорость*)
(*M07KM07_RUN_TIM(IN:= M07KM07_AUX_TIM.Q AND GVL.LRF_AUTO,
				PT:= T#2.15S);*) (*Задержка переключения на малую скорость*)
		//SPEED2 := TRUE;		
(**)IF M07KM07_RUN_TIM.Q AND M07KM07_AUX_TIM.Q THEN
	SPEED2 := TRUE;
END_IF;

IF NOT M07KM07_AUX_TIM.Q THEN
	SPEED2 := FALSE; (*Большая скорость кантователя*)
END_IF;

				
//SPEED2 := M07KM07_RUN_TIM.Q AND M07KM07_AUX_TIM.Q;
IF GVL.LRF_TEST THEN (*Отключение задержки в тестовом режиме*)
	Delay_M07_Run := 0;
ELSE 
	Delay_M07_Run := (GVLR.TIME_M07KM07_DELAY * 1000);
END_IF
		
M07KM07_AUX_TIM(IN:= GVL.M07KM07_AUX,
				PT:= INT_TO_TIME(Delay_M07_Run));				   

GVL.A5_DO_M07KM07_RUN := M07KM07_AUX_TIM.Q; (*Работа/Тормоз Кантователя Выход *)

(*Счетчик циклов Кантователя*)
M07KM07_R_TRIG(CLK := GVL.A5_DO_M07KM07_RUN AND GVL.LRF_AUTO);
IF M07KM07_R_TRIG.Q THEN
	GVLR.PRF_COUNTER_AUTO := GVLR.PRF_COUNTER_AUTO +1;
END_IF


(*GVL.A5_DO_RESERV01 := M07KM07_AUX_TIM.Q AND NOT SPEED2;	(*Большая скорость кантователя*)*)

GVL.A4_DO_XV04KV210 := M07KM07_AUX_TIM.Q AND SPEED2;	(*Малая скорость Кантователя*)
		   
(*Пресс XV01KV207*)
GVL.XV01KV207_ALM := XV01KV207_ALM_TIM.Q OR (GVL.XV01KV207_ALM AND NOT GVL.ALMACK);
XV01KV207_ALM_TIM(IN:= (GVL.A4_DO_XV01KV207 AND NOT SQ05_TIM.Q),
				  PT:= INT_TO_TIME(GVLR.TIME_XV01KV207_ALM *1000));

(*тАЙМЕР ПРИЖИМА*)				  
SQ05_TIM(IN:= GVL.A2_DI_SQ05 (*AND GVL.XV01KV207_AUX*),PT:= REAL_TO_TIME(GVLR.TIMER_SQ5_DELAY * 1000));(*Ввод из MANUAL_FRAME1*)
(*SQ05_TIM(IN:= GVL.A2_DI_SQ05 (*AND GVL.XV01KV207_AUX*),PT:= T#2S);*)
				  
XV01KV207_SUM := GVL.LRFRDYSTS AND GVL.A2_DI_SQ08 AND NOT GVL.A5_DO_M07KM07_RUN AND NOT GVL.A1_DI_M07KM07_ON AND
				 GVL.A2_DI_SQ06 AND NOT GVL.A4_DO_XV03KV209 AND NOT SQ05_TIM.Q;
				 
IF (GVL.A4_DO_XV01KV207 AND GVL.A2_DI_SQ05) OR NOT XV01KV207_SUM OR NOT GVL.LRF_MANUAL THEN
	GVL.XV01KV207_MANOI := FALSE;
END_IF;
				 
GVL.XV01KV207_AUX := (GVL.LRF_TEST AND GVL.XV01KV207_TSTOI AND GVL.A1_DI_SB_TEST AND XV01KV207_SUM) OR 
					 (GVL.LRF_MANUAL AND GVL.XV01KV207_MANOI AND XV01KV207_SUM) OR 
					 (GVL.LRF_AUTO AND XV01KV207_SUM AND GVL.LRFRUNSTS AND A2_DI_SQ08_KEEP AND (GVL.A1_DI_SB_1st_OPER_KEEP OR 
					  GVL.A1_DI_SB_2nd_OPER_KEEP));

XV01KV207_AUX_TIM(IN:= GVL.XV01KV207_AUX AND GVL.A2_DI_M10KM10_ON,
				  PT:= INT_TO_TIME(GVLR.TIME_XV01KV207_DELAY * 1000));
					 
GVL.A4_DO_XV01KV207 := XV01KV207_AUX_TIM.Q;
					 
(*Пресс XV02KV208*)
GVL.XV02KV208_ALM := XV02KV208_ALM_TIM.Q OR (GVL.XV02KV208_ALM AND NOT GVL.ALMACK);
XV02KV208_ALM_TIM(IN:= (GVL.A4_DO_XV02KV208 AND NOT GVL.A2_DI_SQ04),
				  PT:= INT_TO_TIME(GVLR.TIME_XV02KV208_ALM *1000));
				  
				  
XV02KV208_SUM := GVL.LRFRDYSTS AND NOT GVL.A5_DO_M07KM07_RUN AND NOT GVL.A1_DI_M07KM07_ON AND
				 GVL.A2_DI_SQ06 AND NOT GVL.A4_DO_XV03KV209 AND NOT GVL.A2_DI_SQ04;
				 
IF (GVL.A4_DO_XV02KV208 AND GVL.A2_DI_SQ04) OR NOT XV02KV208_SUM OR NOT GVL.LRF_MANUAL THEN
	GVL.XV02KV208_MANOI := FALSE;
END_IF;
				 
GVL.XV02KV208_AUX := (GVL.LRF_TEST AND GVL.XV02KV208_TSTOI AND GVL.A1_DI_SB_TEST AND XV02KV208_SUM) OR 
					 (GVL.LRF_MANUAL AND GVL.XV02KV208_MANOI AND XV02KV208_SUM) OR 
					 (GVL.LRF_AUTO AND XV02KV208_SUM AND GVL.LRFRUNSTS AND NOT A2_DI_SQ08_KEEP);

XV02KV208_AUX_TIM(IN:= GVL.XV02KV208_AUX AND GVL.A2_DI_M10KM10_ON,
				  PT:= INT_TO_TIME(GVLR.TIME_XV02KV208_DELAY * 1000));			 
					 
GVL.A4_DO_XV02KV208 := XV02KV208_AUX_TIM.Q; (*Разжатие пресса*)

(*Маслостанция*)
GVL.M10KM10_ALM := M10KM10_ALM_TIM.Q OR (GVL.M10KM10_ALM AND NOT GVL.ALMACK);
M10KM10_ALM_TIM(IN:= (GVL.A5_DO_M10KM10_RUN AND NOT GVL.A2_DI_M10KM10_ON) OR
					 (NOT GVL.A5_DO_M10KM10_RUN AND GVL.A2_DI_M10KM10_ON),
				PT:= INT_TO_TIME(GVLR.TIME_M10KM10_ALM *1000));
(*				
GVL.PI01_ALM := PI01_ALM_TIM.Q OR (GVL.PI01_ALM AND NOT GVL.ALMACK);
PI01_ALM_TIM(IN:= (GVL.A5_DO_M10KM10_RUN AND NOT GVL.A3_DI_PI01) OR 
				  (GVL.A2_DI_M10KM10_ON AND NOT GVL.A3_DI_PI01),
			 PT:= T#5S);*)

GVL.M10KM10_AUX := GVL.LRFRDYSTS AND (GVL.XV02KV208_AUX OR GVL.XV01KV207_AUX);

GVL.A5_DO_M10KM10_RUN := GVL.M10KM10_AUX;

(*Выталкиватель XV03KV209* Вытолкнуть*)   
GVL.XV03KV209_ALM := XV03KV209_ALM_TIM.Q OR (GVL.XV03KV209_ALM AND NOT GVL.ALMACK);
XV03KV209_ALM_TIM(IN:= (GVL.A4_DO_XV03KV209 AND NOT GVL.A2_DI_SQ07),
				  PT:= INT_TO_TIME(GVLR.TIME_XV03KV209_ALM *1000));
				  
IF (GVL.A2_DI_SQ07 AND GVL.A4_DO_XV03KV209) OR NOT XV03KV209_SUM OR NOT GVL.LRF_MANUAL THEN
	GVL.XV03KV209_MANOI := FALSE;
END_IF;

SQ10_SR(SET1:= NOT GVL.A5_DO_M08KM08_RUN AND NOT GVL.A5_DO_M09UZ09_RUN  AND GVL.A3_DI_SQ10, (*AND NOT GVL.A3_DI_SQ11*)
		RESET:= GVL.A5_DO_M09UZ09_RUN);

XV03KV209_SUM := GVL.LRFRDYSTS AND GVL.A2_DI_SQ08 AND NOT GVL.A5_DO_M07KM07_RUN AND NOT GVL.A1_DI_M07KM07_ON AND
				 NOT GVL.A4_DO_XV01KV207 AND NOT GVL.A4_DO_XV02KV208 AND GVL.A2_DI_SQ05 (*AND 
				 NOT GVL.A3_DI_SQ11 AND GVL.A3_DI_SQ10*);

GVL.XV03KV209_AUX := (GVL.LRF_TEST AND GVL.XV03KV209_TSTOI AND GVL.A1_DI_SB_TEST AND XV03KV209_SUM) OR 
					 (GVL.LRF_MANUAL AND GVL.XV03KV209_MANOI AND XV03KV209_SUM) OR 
					 (GVL.LRF_AUTO AND XV03KV209_SUM AND GVL.LRFRUNSTS AND A2_DI_SQ08_KEEP AND (GVL.A1_DI_SB_1st_OPER_KEEP OR 
					  GVL.A1_DI_SB_2nd_OPER_KEEP) AND SQ10_SR.Q1);
					
XV03KV209_AUX_UP(IN:= GVL.A4_DO_XV03KV209,
				 PT:= INT_TO_TIME(GVLR.TIME_XV03KV209_UP * 1000));
				 
XV03KV209_AUX_TIM(IN:= GVL.XV03KV209_AUX,
				  PT:= INT_TO_TIME(GVLR.TIME_XV03KV209_DELAY * 1000));

GVL.A4_DO_XV03KV209 := XV03KV209_AUX_TIM.Q;

IF GVL.LRF_AUTO AND GVL.LRFRUNSTS AND XV03KV209_AUX_UP.Q AND A2_DI_SQ08_KEEP THEN
	GVL.A1_DI_SB_1st_OPER_KEEP := FALSE;
    GVL.A1_DI_SB_2nd_OPER_KEEP := FALSE;
    A2_DI_SQ08_KEEP := FALSE;
	M09UZ09_READY_TO_RUN := TRUE;
END_IF;

(*M01UZ01_RUN*)	
GVL.M01UZ01_ALM := M01UZ01_ALM_TIM.Q OR (GVL.M01UZ01_ALM AND NOT GVL.ALMACK);
M01UZ01_ALM_TIM(IN:= (GVL.A5_DO_M01UZ01_RUN AND NOT GVL.A1_DI_M01UZ01_ON) OR
					 (GVL.A1_DI_M01UZ01_ON AND NOT GVL.A5_DO_M01UZ01_RUN),
				PT:= INT_TO_TIME(GVLR.TIME_M01UZ01_ALM *1000));
		  				  
M01UZ01_SUM := GVL.LRFRDYSTS AND GVL.M01UZ01_CFGOI;

IF NOT GVL.LRF_MANUAL THEN
	GVL.M01UZ01_MANOI := FALSE;
END_IF;

GVL.M01UZ01_AUX := (GVL.LRF_TEST AND GVL.M01UZ01_TSTOI AND GVL.A1_DI_SB_TEST AND M01UZ01_SUM) OR
				   (GVL.LRF_MANUAL AND GVL.M01UZ01_MANOI AND M01UZ01_SUM) OR 
				   (GVL.LRF_AUTO AND GVL.LRFRUNSTS AND GVL.A1_DI_M03UZ03_ON AND M01UZ01_SUM);

M01UZ01_AUX_TIM(IN:= GVL.M01UZ01_AUX, 
				PT:= INT_TO_TIME(GVLR.TIME_M01UZ01_DELAY * 1000));
				   
GVL.A5_DO_M01UZ01_RUN := M01UZ01_AUX_TIM.Q;

(*M02UZ02_RUN*)	(*Обсыпной бункер резервный*)

(*Резчик*)
GVL.RESET_SQ2_CNT := NOT GVL.A1_DI_M04KM04_ON;
GVL.A2_DI_SQ02_CLON := GVL.A2_DI_SQ02_CNT > 0;

(*TON_SQ15(IN := GVL.A2_DI_SQ15, PT := T#100MS);(*Задержка запуска Резчика*)*)
TON_SQ15(IN := NOT GVL.A1_DI_M04KM04_ON, PT := T#200MS);(*Задержка запуска Резчика после останова*)

A2_DI_SQ02_OSR(CLK:= GVL.A2_DI_SQ02_CLON);
(*A2_DI_SQ15_OSR(CLK:= GVL.A2_DI_SQ15 AND NOT GVL.A1_DI_M04KM04_ON);	*)
(*A2_DI_SQ15_OSR(CLK:= TON_SQ15.Q AND NOT GVL.A1_DI_M04KM04_ON);*)		
SQ15_QSR(CLK :=	GVL.A2_DI_SQ15);  (*Нарастание Запуск резчика*)
A2_DI_SQ15_OSR(CLK:= TON_SQ15.Q AND SQ15_QSR.Q); 		  				  


	  				  
M02UZ02_SUM := GVL.LRFRDYSTS;

IF A2_DI_SQ02_OSR.Q OR NOT GVL.LRF_MANUAL THEN
	GVL.M02UZ02_MANOI := FALSE;
END_IF;

M02UZ02_SR(SET1:= (GVL.LRF_TEST AND GVL.M02UZ02_TSTOI AND GVL.A1_DI_SB_TEST) OR (GVL.LRF_AUTO AND A2_DI_SQ15_OSR.Q AND GVL.LRFRUNSTS (*AND GVL.A3_DI_KV301*)) OR
				  (GVL.LRF_MANUAL AND GVL.M02UZ02_MANOI), 
		   RESET:= A2_DI_SQ02_OSR.Q OR GVL.A1_DI_SB_STOP, (*Останов резчика концевиком и кнопкой стоп*)
		   Q1=> M02UZ02_START);

GVL.M02UZ02_AUX := (GVL.LRF_TEST AND M02UZ02_START AND M02UZ02_SUM) OR
				   (GVL.LRF_MANUAL AND GVL.M02UZ02_MANOI AND M02UZ02_SUM AND M02UZ02_START) OR
				   (GVL.LRF_AUTO AND GVL.LRFRUNSTS AND M02UZ02_START AND M02UZ02_SUM); 

M02UZ02_AUX_TIM(IN:= GVL.M02UZ02_AUX, 
				PT:= INT_TO_TIME(GVLR.TIME_M02UZ02_DELAY * 1000));
		   
GVL.A5_DO_M02UZ02_RUN_FORW := M02UZ02_AUX_TIM.Q ;
GVL.A5_DO_M04KM04_RUN := M02UZ02_AUX_TIM.Q;
				  
(*M03UZ03_RUN*)	(*Транспортер резчиковый*)
GVL.M03UZ03_ALM := M03UZ03_ALM_TIM.Q OR (GVL.M03UZ03_ALM AND NOT GVL.ALMACK);
M03UZ03_ALM_TIM(IN:= (GVL.A5_DO_M03UZ03_RUN AND NOT GVL.A1_DI_M03UZ03_ON) OR
					 (GVL.A1_DI_M03UZ03_ON AND NOT GVL.A5_DO_M03UZ03_RUN),
				PT:= INT_TO_TIME(GVLR.TIME_M03UZ03_ALM *1000));
		  				  
M03UZ03_SUM := GVL.LRFRDYSTS AND GVL.M03UZ03_CFGOI;

IF NOT GVL.LRF_MANUAL THEN
	GVL.M03UZ03_MANOI := FALSE;
END_IF;

GVL.M03UZ03_AUX := (GVL.LRF_TEST AND GVL.M03UZ03_TSTOI AND GVL.A1_DI_SB_TEST AND M03UZ03_SUM) OR
				   (GVL.LRF_MANUAL AND GVL.M03UZ03_MANOI AND M03UZ03_SUM) OR 
				   (GVL.LRF_AUTO AND GVL.LRFRUNSTS AND (GVL.A1_DI_M05UZ05_ON OR NOT GVL.M05UZ05_CFGOI) AND M03UZ03_SUM);

M03UZ03_AUX_TIM(IN:= GVL.M03UZ03_AUX, 
				PT:= INT_TO_TIME(GVLR.TIME_M03UZ03_DELAY * 1000));
				   
GVL.A5_DO_M03UZ03_RUN := M03UZ03_AUX_TIM.Q;

(*M05UZ05_RUN*)	(*Транспортер угловой*)	
GVL.M05UZ05_ALM := M05UZ05_ALM_TIM.Q OR (GVL.M05UZ05_ALM AND NOT GVL.ALMACK);
M05UZ05_ALM_TIM(IN:= (GVL.A5_DO_M05UZ05_RUN AND NOT GVL.A1_DI_M05UZ05_ON) OR
					 (GVL.A1_DI_M05UZ05_ON AND NOT GVL.A5_DO_M05UZ05_RUN),
				PT:= INT_TO_TIME(GVLR.TIME_M05UZ05_ALM *1000));
		  
M05UZ05_SUM := GVL.LRFRDYSTS AND NOT GVL.A2_DI_SQ03 AND GVL.M05UZ05_CFGOI;

IF NOT GVL.LRF_MANUAL THEN
	GVL.M05UZ05_MANOI := FALSE;
END_IF;

GVL.M05UZ05_AUX := (GVL.LRF_TEST AND GVL.M05UZ05_TSTOI AND GVL.A1_DI_SB_TEST AND M05UZ05_SUM) OR
				   (GVL.LRF_MANUAL AND GVL.M05UZ05_MANOI AND M05UZ05_SUM) OR 
				   (GVL.LRF_AUTO AND GVL.LRFRUNSTS AND (GVL.A1_DI_M06UZ06_ON OR NOT GVL.M06UZ06_CFGOI) AND M05UZ05_SUM);

M05UZ05_AUX_TIM(IN:= GVL.M05UZ05_AUX, 
				PT:= INT_TO_TIME(GVLR.TIME_M05UZ05_DELAY * 1000));
				   
GVL.A5_DO_M05UZ05_RUN := M05UZ05_AUX_TIM.Q;

(*M06UZ06_RUN*)	(*Подающий транспортер*)
GVL.M06UZ06_ALM := M06UZ06_ALM_TIM.Q OR (GVL.M06UZ06_ALM AND NOT GVL.ALMACK);
M06UZ06_ALM_TIM(IN:= (GVL.A5_DO_M06UZ06_RUN AND NOT GVL.A1_DI_M06UZ06_ON) OR
					 (GVL.A1_DI_M06UZ06_ON AND NOT GVL.A5_DO_M06UZ06_RUN),
				PT:= INT_TO_TIME(GVLR.TIME_M06UZ06_ALM *1000));
		  				  
M06UZ06_SUM := GVL.LRFRDYSTS AND NOT GVL.A2_DI_SQ03 AND GVL.M06UZ06_CFGOI;

IF NOT GVL.LRF_MANUAL THEN
	GVL.M06UZ06_MANOI := FALSE;
END_IF;

GVL.M06UZ06_AUX := (GVL.LRF_TEST AND GVL.M06UZ06_TSTOI AND GVL.A1_DI_SB_TEST AND M06UZ06_SUM) OR
				   (GVL.LRF_MANUAL AND GVL.M06UZ06_MANOI AND M06UZ06_SUM) OR 
				   (GVL.LRF_AUTO AND GVL.LRFRUNSTS AND M06UZ06_SUM);

M06UZ06_AUX_TIM(IN:= GVL.M06UZ06_AUX, 
				PT:= INT_TO_TIME(GVLR.TIME_M06UZ06_DELAY * 1000));
				   
GVL.A5_DO_M06UZ06_RUN := M06UZ06_AUX_TIM.Q;			  
GVL.A5_DO_M13KM13_RUN := GVL.A5_DO_M06UZ06_RUN; (*Доп тр-р на KM13*)

(*M08KM08_RUN*)	(*Палетный транспортер*)
GVL.M08KM08_ALM := M08KM08_ALM_TIM.Q OR (GVL.M08KM08_ALM AND NOT GVL.ALMACK);
M08KM08_ALM_TIM(IN:= (GVL.A5_DO_M08KM08_RUN AND NOT GVL.A1_DI_M08KM08_ON) OR
					 (GVL.A1_DI_M08KM08_ON AND NOT GVL.A5_DO_M08KM08_RUN),
				PT:= INT_TO_TIME(GVLR.TIME_M08KM08_ALM *1000));
		  				  
M08KM08_SUM := GVL.LRFRDYSTS;

IF NOT GVL.LRF_MANUAL THEN
	GVL.M08KM08_MANOI := FALSE;
END_IF;

M08KM08_SR(SET1:= (GVL.LRF_AUTO AND GVL.LRFRUNSTS AND NOT GVL.A2_DI_M09UZ09_ON AND NOT GVL.A3_DI_SQ10), 
		   RESET:= M08KM08_AUX_OFF.Q OR NOT GVL.LRFRUNSTS);

GVL.M08KM08_AUX := (GVL.LRF_TEST AND GVL.M08KM08_TSTOI AND GVL.A1_DI_SB_TEST AND M08KM08_SUM) OR
				   (GVL.LRF_MANUAL AND GVL.M08KM08_MANOI AND M08KM08_SUM) OR 
				   (GVL.LRF_AUTO AND GVL.LRFRUNSTS AND M08KM08_SR.Q1 (*AND NOT GVL.A3_DI_SQ11*) AND M08KM08_SUM);

M08KM08_AUX_TIM(IN:= GVL.M08KM08_AUX, 
				PT:= INT_TO_TIME(GVLR.TIME_M08KM08_DELAY * 1000));

M08KM08_AUX_OFF(IN:= (GVL.LRF_AUTO AND GVL.LRFRUNSTS AND GVL.A1_DI_M08KM08_ON), 
				PT:= INT_TO_TIME(GVLR.TIME_M08KM08_OFF * 1000));
				   
GVL.A5_DO_M08KM08_RUN := M08KM08_AUX_TIM.Q;

(*M09UZ09_RUN*) (*Выгружной транспортер*)
GVL.M09UZ09_ALM := M09UZ09_ALM_TIM.Q OR (GVL.M09UZ09_ALM AND NOT GVL.ALMACK);
M09UZ09_ALM_TIM(IN:= (GVL.A5_DO_M09UZ09_RUN AND NOT GVL.A2_DI_M09UZ09_ON) OR
					 (GVL.A2_DI_M09UZ09_ON AND NOT GVL.A5_DO_M09UZ09_RUN),
				PT:= INT_TO_TIME(GVLR.TIME_M09UZ09_ALM *1000));	

GVL.A2_DI_SQ06_ALM := A2_DI_SQ06_ALM_TIM.Q OR (GVL.A2_DI_SQ06_ALM AND NOT GVL.ALMACK);			
A2_DI_SQ06_ALM_TIM(IN:= NOT GVL.A2_DI_SQ06 AND GVL.LRFRDYSTS,
				   PT:= INT_TO_TIME(GVLR.TIME_SQ06_ALM *1000));	
		  				  
M09UZ09_SUM := GVL.LRFRDYSTS;

IF NOT GVL.LRF_MANUAL THEN
	GVL.M09UZ09_MANOI := FALSE;
END_IF;

(*A3_DI_SQ11_TIM(IN:= GVL.A3_DI_SQ11, 
			   PT:= T#1.5S);*)

M09UZ09_SR(SET1:= (GVL.LRF_AUTO AND GVL.LRFRUNSTS (*AND A3_DI_SQ11_TIM.Q*) AND 
				   (*NOT GVL.A1_DI_SB_1st_OPER_KEEP AND NOT GVL.A1_DI_SB_2nd_OPER_KEEP AND*) M09UZ09_READY_TO_RUN), 
		   RESET:= M09UZ09_AUX_OFF.Q OR NOT GVL.LRFRUNSTS, 
		   Q1=> M09UZ09_START);

GVL.M09UZ09_AUX := (GVL.LRF_TEST AND GVL.M09UZ09_TSTOI AND GVL.A1_DI_SB_TEST AND M09UZ09_SUM) OR
				   (GVL.LRF_MANUAL AND GVL.M09UZ09_MANOI AND M09UZ09_SUM) OR 
				   (GVL.LRF_AUTO AND GVL.LRFRUNSTS AND NOT GVL.A1_DI_M08KM08_ON AND M09UZ09_START AND M09UZ09_SUM AND GVL.A2_DI_SQ06 AND 
					M09UZ09_READY_TO_RUN);

M09UZ09_AUX_TIM(IN:= GVL.M09UZ09_AUX, 
				PT:= INT_TO_TIME(GVLR.TIME_M09UZ09_DELAY * 1000));
				
M09UZ09_AUX_OFF(IN:= (GVL.LRF_AUTO AND GVL.LRFRUNSTS AND GVL.A2_DI_M09UZ09_ON )(*AND NOT GVL.A3_DI_SQ11*),
				PT:= INT_TO_TIME(GVLR.TIME_M09UZ09_OFF * 1000));

IF M09UZ09_AUX_OFF.Q THEN
	M09UZ09_READY_TO_RUN := FALSE;
END_IF;
				   
GVL.A5_DO_M09UZ09_RUN := M09UZ09_AUX_TIM.Q;

(*M14UZ14_RUN*)
GVL.M14UZ14_ALM := M14UZ14_ALM_TIM.Q OR (GVL.M14UZ14_ALM AND NOT GVL.ALMACK);
M14UZ14_ALM_TIM(IN:= (GVL.A5_DO_M14UZ14_RUN AND NOT GVL.A2_DI_M14UZ14_ON) OR
					 (GVL.A2_DI_M14UZ14_ON AND NOT GVL.A5_DO_M14UZ14_RUN),
				PT:= INT_TO_TIME(GVLR.TIME_M14UZ14_ALM *1000));	
		  				  
M14UZ14_SUM := GVL.LRFRDYSTS AND GVL.M14UZ14_CFGOI AND NOT GVL.A3_DI_KV302;

IF NOT GVL.LRF_MANUAL THEN
	GVL.M14UZ14_MANOI := FALSE;
END_IF;

M14UZ14_SR(SET1:= (GVL.LRF_AUTO AND GVL.LRFRUNSTS AND GVL.A2_DI_M09UZ09_ON), 
		   RESET:= M14UZ14_AUX_OFF.Q OR NOT GVL.LRFRUNSTS);

GVL.M14UZ14_AUX := (GVL.LRF_TEST AND GVL.M14UZ14_TSTOI AND GVL.A1_DI_SB_TEST AND M14UZ14_SUM) OR
				   (GVL.LRF_MANUAL AND GVL.M14UZ14_MANOI AND M14UZ14_SUM) OR 
				   (GVL.LRF_AUTO AND GVL.LRFRUNSTS AND M14UZ14_SR.Q1 AND M14UZ14_SUM);

M14UZ14_AUX_TIM(IN:= GVL.M14UZ14_AUX, 
				PT:= INT_TO_TIME(GVLR.TIME_M14UZ14_DELAY * 1000));
				
M14UZ14_AUX_OFF(IN:= (GVL.LRF_AUTO AND GVL.LRFRUNSTS AND GVL.A2_DI_M14UZ14_ON), 
				PT:= INT_TO_TIME(GVLR.TIME_M14UZ14_OFF * 1000));
				
GVL.A5_DO_M14UZ14_RUN := M14UZ14_AUX_TIM.Q;

(*M11KM11_RUN*)	
GVL.M11KM11_ALM := M11KM11_ALM_TIM.Q OR (GVL.M11KM11_ALM AND NOT GVL.ALMACK);
M11KM11_ALM_TIM(IN:= (GVL.A5_DO_M11KM11_RUN AND NOT GVL.A2_DI_M11KM11_ON) OR
					 (GVL.A2_DI_M11KM11_ON AND NOT GVL.A5_DO_M11KM11_RUN),
				PT:= INT_TO_TIME(GVLR.TIME_M11KM11_ALM *1000));
		  				  
M11KM11_SUM := GVL.LRFRDYSTS AND GVL.M11KM11_CFGOI;

IF NOT GVL.LRF_MANUAL THEN
	GVL.M11KM11_MANOI := FALSE;
END_IF;

GVL.M11KM11_AUX := (GVL.LRF_TEST AND GVL.M11KM11_TSTOI AND GVL.A1_DI_SB_TEST AND M11KM11_SUM) OR
				   (GVL.LRF_MANUAL AND GVL.M11KM11_MANOI AND M11KM11_SUM) OR 
				   (GVL.LRF_AUTO AND GVL.LRFRUNSTS AND M11KM11_SUM);

M11KM11_AUX_TIM(IN:= GVL.M11KM11_AUX, 
				PT:= INT_TO_TIME(GVLR.TIME_M11KM11_DELAY * 1000));
				   
GVL.A5_DO_M11KM11_RUN := M11KM11_AUX_TIM.Q;

(*M12KM12_RUN*)	
GVL.M12KM12_ALM := M12KM12_ALM_TIM.Q OR (GVL.M12KM12_ALM AND NOT GVL.ALMACK);
M12KM12_ALM_TIM(IN:= (GVL.A5_DO_M12KM12_RUN AND NOT GVL.A2_DI_M12KM12_ON) OR
					 (GVL.A2_DI_M12KM12_ON AND NOT GVL.A5_DO_M12KM12_RUN),
				PT:= INT_TO_TIME(GVLR.TIME_M12KM12_ALM *1000));
		  				  
M12KM12_SUM := GVL.LRFRDYSTS AND GVL.M12KM12_CFGOI;

IF NOT GVL.LRF_MANUAL THEN
	GVL.M12KM12_MANOI := FALSE;
END_IF;

GVL.M12KM12_AUX := (GVL.LRF_TEST AND GVL.M12KM12_TSTOI AND GVL.A1_DI_SB_TEST AND M12KM12_SUM) OR
				   (GVL.LRF_MANUAL AND GVL.M12KM12_MANOI AND M12KM12_SUM) OR 
				   (GVL.LRF_AUTO AND GVL.LRFRUNSTS AND GVL.A1_DI_M06UZ06_ON AND M12KM12_SUM);

M12KM12_AUX_TIM(IN:= GVL.M12KM12_AUX, 
				PT:= INT_TO_TIME(GVLR.TIME_M12KM12_DELAY * 1000));
				   
GVL.A5_DO_M12KM12_RUN := M12KM12_AUX_TIM.Q;

(*MV01KM00_RUN*)
GVL.MV01KM00_ALM := MV01KM00_ALM_TIM.Q OR (GVL.MV01KM00_ALM AND NOT GVL.ALMACK);
MV01KM00_ALM_TIM(IN:= (GVL.A5_DO_MV01KM00_RUN AND NOT GVL.A1_DI_MV01KM00_ON) OR
					 (GVL.A1_DI_MV01KM00_ON AND NOT GVL.A5_DO_MV01KM00_RUN),
				PT:= INT_TO_TIME(GVLR.TIME_MV01KM00_ALM *1000));
		  				  
MV01KM00_SUM := GVL.LRFRDYSTS AND GVL.MV01KM00_CFGOI;

IF NOT GVL.LRF_MANUAL THEN
	GVL.MV01KM00_MANOI := FALSE;
END_IF;

GVL.MV01KM00_AUX := (GVL.LRF_TEST AND GVL.MV01KM00_TSTOI AND GVL.A1_DI_SB_TEST AND MV01KM00_SUM) OR
				   (GVL.LRF_MANUAL AND GVL.MV01KM00_MANOI AND MV01KM00_SUM) OR
				   (GVL.LRF_AUTO AND GVL.LRFRUNSTS AND MV01KM00_IMP.OUT);
				   
MV01KM00_IMP(ENABLE:= GVL.LRF_AUTO AND GVL.LRFRUNSTS AND GVL.MV01KM00_CFGOI, 
			 TIMELOW:= INT_TO_TIME(GVLR.TIME_MV01KM00_ON * 1000), 
			 TIMEHIGH:= INT_TO_TIME(GVLR.TIME_MV01KM00_OFF * 1000));
				   
GVL.A5_DO_MV01KM00_RUN := GVL.MV01KM00_AUX;

END_PROGRAM

// Device/Application/SEQUENSER
PROGRAM SEQUENSER
VAR
	PRF_SHIFT_STEP_OSR : R_TRIG;
END_VAR


(*Этапы


GVLR.PRF_SHIFT_STEP := NOT GVLR.PRF_SHIFT_STEP AND  (GVLR.PRF_STEP1 AND (MAIN.A1_DI_SB_1st_OPER_KEEP OR MAIN.A1_DI_SB_2nd_OPER_KEEP) AND 
													 NOT MOTORS.A2_DI_SQ08_KEEP AND GVL.LRF_AUTO) OR
											   		(GVLR.PRF_STEP2 AND ) OR
											   		(GVLR.PRF_STEP3 AND ) OR
											   		(GVLR.PRF_STEP4 AND ) OR
											   		(GVLR.PRF_STEP5 AND ) OR
											   		(GVLR.PRF_STEP6 AND );
PRF_SHIFT_STEP_OSR(CLK:= GVLR.PRF_SHIFT_STEP);

IF PRF_SHIFT_STEP_OSR.Q AND GVL.LRF_AUTO THEN
	GVLR.PRF_STEPS := GVLR.PRF_STEPS + 1;
END_IF;											   
(**)
GVLR.PRF_STEP1 := GVLR.PRF_STEPS = 1;
GVLR.PRF_STEP2 := GVLR.PRF_STEPS = 2;
GVLR.PRF_STEP3 := GVLR.PRF_STEPS = 3;
GVLR.PRF_STEP4 := GVLR.PRF_STEPS = 4;
GVLR.PRF_STEP5 := GVLR.PRF_STEPS = 5;
GVLR.PRF_STEP6 := GVLR.PRF_STEPS = 6;*)

END_PROGRAM

// Device/Application/TEST_FRAME_2
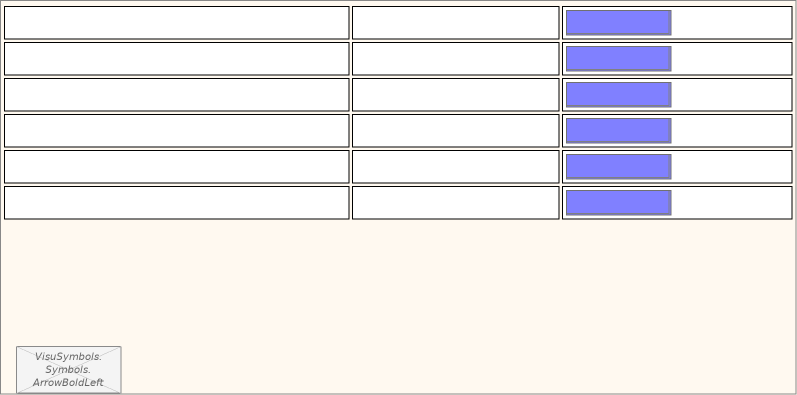
VISUALIZATION TEST_FRAME_2  // 797x395
    Image (16,346 105x47), image: VisuSymbols.Symbols.ArrowBoldLeft
        OnMouseClick: FrameSelectionChange Selection=Selection=-1, GlobSel=IndExpr=4, AssignDir=Main.GenElemInst_39, AssignType=Directly, SelType=Globally
    Rectangle (4,6 345x33), text list: 'IM', text index: 12
    Rectangle (352,6 207x33), text list: 'IM_TAGS', text index: 10
    Rectangle (562,6 230x33)
    Button (566,10 105x25), colour toggle: GVL.M08KM08_TSTOI
        OnMouseClick: execute { GVL.TSTOI := 12; }
    Rectangle (4,42 345x33), text list: 'IM', text index: 13
    Rectangle (4,78 345x33), text list: 'IM', text index: 14
    Rectangle (4,114 345x33), text list: 'IM', text index: 15
    Rectangle (4,150 345x33), text list: 'IM', text index: 16
    Rectangle (4,186 345x33), text list: 'IM', text index: 17
    Rectangle (352,42 207x33), text list: 'IM_TAGS', text index: 11
    Rectangle (352,78 207x33), text list: 'IM_TAGS', text index: 12
    Rectangle (352,114 207x33), text list: 'IM_TAGS', text index: 13
    Rectangle (352,150 207x33), text list: 'IM_TAGS', text index: 14
    Rectangle (352,186 207x33), text list: 'IM_TAGS', text index: 15
    Rectangle (562,42 230x33)
    Button (566,46 105x25), colour toggle: GVL.M09UZ09_TSTOI
        OnMouseClick: execute { GVL.TSTOI := 13; }
    Rectangle (562,78 230x33)
    Button (566,82 105x25), colour toggle: GVL.M10KM10_TSTOI
        OnMouseClick: execute { GVL.TSTOI := 14; }
    Rectangle (562,114 230x33)
    Button (566,118 105x25), colour toggle: GVL.M11KM11_TSTOI
        OnMouseClick: execute { GVL.TSTOI := 15; }
    Rectangle (562,150 230x33)
    Button (566,154 105x25), colour toggle: GVL.M12KM12_TSTOI
        OnMouseClick: execute { GVL.TSTOI := 16; }
    Rectangle (562,186 230x33)
    Button (566,190 105x25), colour toggle: GVL.M14UZ14_TSTOI
        OnMouseClick: execute { GVL.TSTOI := 17; }
END_VISUALIZATION

// Device/Application/SETTINGS_FRAME
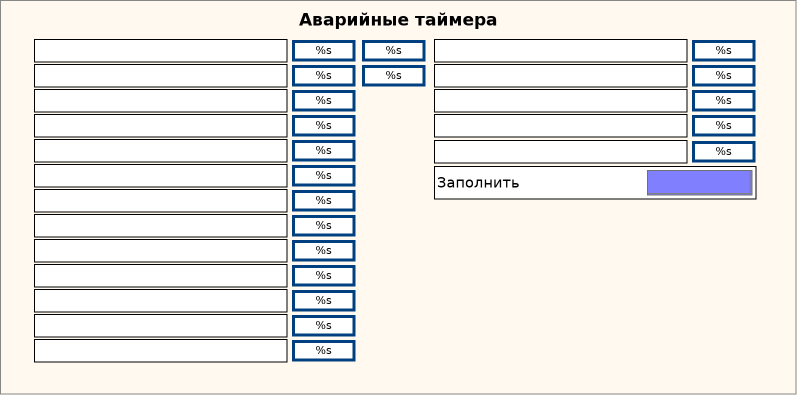
VISUALIZATION SETTINGS_FRAME  // 797x395
    Rectangle (292,40 63x21), "%s", text variable: GVLR.TIME_XV01KV207_ALM
        OnMouseClick: write the text variable via VisuDialogs.Numpad
    Rectangle (34,39 253x23), text list: 'IM', text index: 1
    Rectangle (34,64 253x23), text list: 'IM', text index: 3
    Rectangle (34,89 253x23), text list: 'IM', text index: 5
    Rectangle (34,114 253x23), text list: 'IM', text index: 6
    Rectangle (34,139 253x23), text list: 'IM', text index: 7
    Rectangle (34,164 253x23), text list: 'IM', text index: 8
    Rectangle (34,189 253x23), text list: 'IM', text index: 9
    Rectangle (34,214 253x23), text list: 'IM', text index: 10
    Rectangle (34,239 253x23), text list: 'IM', text index: 11
    Rectangle (34,264 253x23), text list: 'IM', text index: 12
    Rectangle (34,289 253x23), text list: 'IM', text index: 13
    Rectangle (34,314 253x23), text list: 'IM', text index: 14
    Rectangle (34,339 253x23), text list: 'IM', text index: 15
    Rectangle (434,39 253x23), text list: 'IM', text index: 16
    Rectangle (434,64 253x23), text list: 'IM', text index: 17
    Rectangle (362,40 63x21), "%s", text variable: GVLR.TIME_XV02KV208_ALM
        OnMouseClick: write the text variable via VisuDialogs.Numpad
    Rectangle (292,65 63x21), "%s", text variable: GVLR.TIME_XV03KV209_ALM
        OnMouseClick: write the text variable via VisuDialogs.Numpad
    Rectangle (362,65 63x21), "%s", text variable: GVLR.TIME_XV04KV210_ALM
        OnMouseClick: write the text variable via VisuDialogs.Numpad
    Rectangle (292,90 63x21), "%s", text variable: GVLR.TIME_MV01KM00_ALM
        OnMouseClick: write the text variable via VisuDialogs.Numpad
    Rectangle (292,115 63x21), "%s", text variable: GVLR.TIME_M01UZ01_ALM
        OnMouseClick: write the text variable via VisuDialogs.Numpad
    Rectangle (292,140 63x21), "%s", text variable: GVLR.TIME_M03UZ03_ALM
        OnMouseClick: write the text variable via VisuDialogs.Numpad
    Rectangle (292,165 63x21), "%s", text variable: GVLR.TIME_M04KM04_ALM
        OnMouseClick: write the text variable via VisuDialogs.Numpad
    Rectangle (292,190 63x21), "%s", text variable: GVLR.TIME_M05UZ05_ALM
        OnMouseClick: write the text variable via VisuDialogs.Numpad
    Rectangle (292,215 63x21), "%s", text variable: GVLR.TIME_M06UZ06_ALM
        OnMouseClick: write the text variable via VisuDialogs.Numpad
    Rectangle (292,240 63x21), "%s", text variable: GVLR.TIME_M07KM07_ALM
        OnMouseClick: write the text variable via VisuDialogs.Numpad
    Rectangle (292,265 63x21), "%s", text variable: GVLR.TIME_M08KM08_ALM
        OnMouseClick: write the text variable via VisuDialogs.Numpad
    Rectangle (292,290 63x21), "%s", text variable: GVLR.TIME_M09UZ09_ALM
        OnMouseClick: write the text variable via VisuDialogs.Numpad
    Rectangle (292,315 63x21), "%s", text variable: GVLR.TIME_M10KM10_ALM
        OnMouseClick: write the text variable via VisuDialogs.Numpad
    Rectangle (292,340 63x21), "%s", text variable: GVLR.TIME_M11KM11_ALM
        OnMouseClick: write the text variable via VisuDialogs.Numpad
    Rectangle (692,40 63x21), "%s", text variable: GVLR.TIME_M12KM12_ALM
        OnMouseClick: write the text variable via VisuDialogs.Numpad
    Rectangle (692,65 63x21), "%s", text variable: GVLR.TIME_M14UZ14_ALM
        OnMouseClick: write the text variable via VisuDialogs.Numpad
    Rectangle (0,2 797x35), "Аварийные таймера"
    Rectangle (434,89 253x23), text list: 'IM', text index: 18
    Rectangle (434,114 253x23), text list: 'IM', text index: 19
    Rectangle (692,90 63x21), "%s", text variable: GVLR.TIME_PI01_ALM
        OnMouseClick: write the text variable via VisuDialogs.Numpad
    Rectangle (692,115 63x21), "%s", text variable: GVLR.TIME_SQ08_ALM
        OnMouseClick: write the text variable via VisuDialogs.Numpad
    Line (450,41)
    Rectangle (434,166 322x33), "Заполнить"
    Button (647,170 105x25), colour toggle: Main.SET_SETTINGS
        OnMouseDown: execute { Main.SET_SETTINGS := TRUE; }
        OnMouseUp: execute { Main.SET_SETTINGS := FALSE; }
    Rectangle (434,140 253x23), text list: 'IM', text index: 20
    Rectangle (692,141 63x21), "%s", text variable: GVLR.TIME_SQ06_ALM
        OnMouseClick: write the text variable via VisuDialogs.Numpad
END_VISUALIZATION

// Device/Application/PRF_FRAME
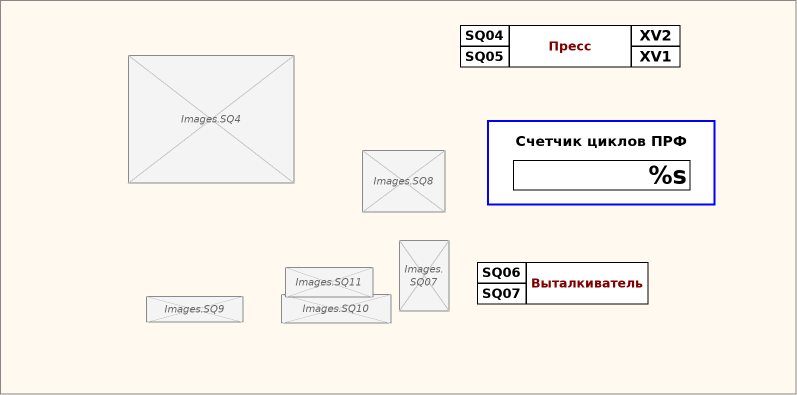
VISUALIZATION PRF_FRAME  // 797x395, background image Images.PRF
    Image (399,240 50x71), invisible if: NOT GVL.A2_DI_SQ06, image: Images.SQ06
    Image (399,240 50x71), invisible if: NOT GVL.A2_DI_SQ07, image: Images.SQ07
    Image (128,55 166x128), invisible if: NOT GVL.A2_DI_SQ05, image: Images.SQ5
    Image (128,55 166x128), invisible if: NOT GVL.A2_DI_SQ04, image: Images.SQ4
    Image (146,296 97x26), invisible if: NOT GVL.A2_DI_SQ09, image: Images.SQ9
    Image (281,294 110x29), invisible if: NOT GVL.A3_DI_SQ10, image: Images.SQ10
    Image (362,150 83x62), invisible if: NOT GVL.A2_DI_SQ08, image: Images.SQ8
    Rectangle (460,25 49x21), "SQ04"
    Rectangle (460,46 49x21), "SQ05"
    Rectangle (477,262 49x21), "SQ06"
    Rectangle (477,283 49x21), "SQ07"
    Rectangle (526,262 122x42), "Выталкиватель"
    Rectangle (509,25 122x42), "Пресс", colour toggle: GVL.A5_DO_M10KM10_RUN
    Image (285,267 88x30), invisible if: NOT GVL.A3_DI_SQ11, image: Images.SQ11
    Group (487,120 228x85)
        RoundedRectangle (0,0 228x85)
        Rectangle (26,40 177x30), "%s", text variable: GVLR.PRF_COUNTER_AUTO
        Rectangle (26,6 177x30), "Счетчик циклов ПРФ"
    Rectangle (631,25 49x21), "XV2", colour toggle: GVL.A4_DO_XV02KV208
    Rectangle (631,46 49x21), "XV1", colour toggle: GVL.A4_DO_XV01KV207
END_VISUALIZATION

// Device/Application/ALARM_FRAME
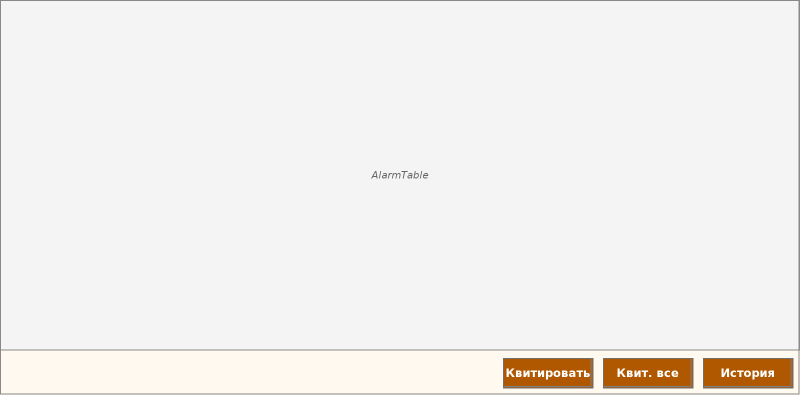
VISUALIZATION ALARM_FRAME  // 800x395
VAR_IN_OUT
END_VAR
VAR
	bAckSel : BOOL;
	bAckVisible : BOOL;
	bHistory : BOOL;
	bFreezeScrlPos : BOOL;
END_VAR
    AlarmTable (0,0 800x350)
        Column[0]: ColumnTitle=Время
        Column[1]: ColumnTitle=Сообщение
        Column[2]: ColumnTitle=Время квитирования
        p1521930926: __All
        p1663851261: __All
        p428520879: bAckSel
        p2607059081: bAckVisible
        p3266827225: bHistory
        p3894972949: bFreezeScrlPos
    Button (503,358 90x30), "Квитировать"
        toggle bAckSel
    Button (603,358 90x30), "Квит. все"
        toggle bAckVisible
    Button (703,358 90x30), "История"
        toggle bHistory
END_VISUALIZATION

// Device/Application/MODE_FRAME
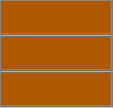
VISUALIZATION MODE_FRAME  // 113x108
    Button (0,72 113x35), text list: 'Mode', text index: 1
        OnMouseClick: execute { GVL.LRF_MODE:=1; }
        OnMouseClick:  Dialog=MODE_FRAME, Result=OK, NumpadKeypadSet=True
    Button (0,36 113x35), text list: 'Mode', text index: 2
        OnMouseClick: execute { GVL.LRF_MODE:=2; }
        OnMouseClick:  Dialog=MODE_FRAME, Result=OK, NumpadKeypadSet=True
        OnMouseClick: FrameSelectionChange Selection=Selection=-1, GlobSel=IndExpr=4, AssignDir=Main.GenElemInst_39, AssignType=Directly, SelType=Globally
    Button (0,0 113x35), text list: 'Mode', text index: 3
        OnMouseClick: execute { GVL.LRF_MODE:=3; }
        OnMouseClick:  Dialog=MODE_FRAME, Result=OK, NumpadKeypadSet=True
END_VISUALIZATION

// Device/Application/TEST_FRAME_1
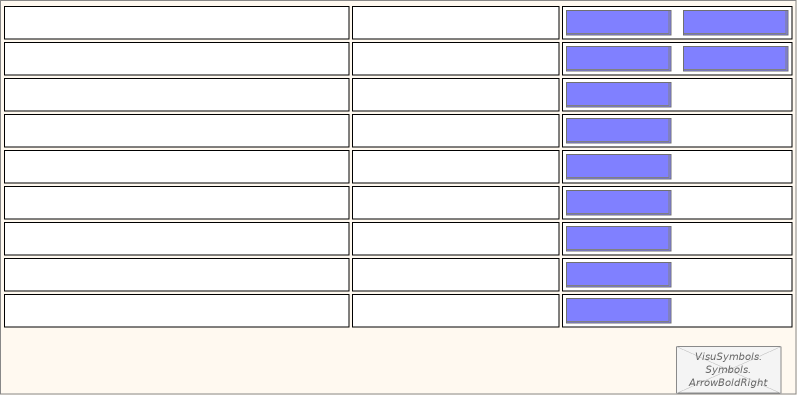
VISUALIZATION TEST_FRAME_1  // 797x395
    Rectangle (4,6 345x33), text list: 'IM', text index: 1
    Rectangle (352,6 207x33), text list: 'IM_TAGS', text index: 1
    Rectangle (562,6 230x33)
    Button (566,10 105x25), colour toggle: GVL.XV01KV207_TSTOI
        OnMouseClick: execute { GVL.TSTOI := 1; }
    Button (683,10 105x25), colour toggle: GVL.XV02KV208_TSTOI
        OnMouseClick: execute { GVL.TSTOI := 2; }
    Rectangle (4,42 345x33), text list: 'IM', text index: 3
    Rectangle (4,78 345x33), text list: 'IM', text index: 5
    Rectangle (4,114 345x33), text list: 'IM', text index: 6
    Rectangle (4,150 345x33), text list: 'IM', text index: 7
    Rectangle (4,186 345x33), text list: 'IM', text index: 8
    Rectangle (4,222 345x33), text list: 'IM', text index: 9
    Rectangle (4,258 345x33), text list: 'IM', text index: 10
    Rectangle (4,294 345x33), text list: 'IM', text index: 11
    Rectangle (352,42 207x33), text list: 'IM_TAGS', text index: 2
    Rectangle (352,78 207x33), text list: 'IM_TAGS', text index: 3
    Rectangle (352,114 207x33), text list: 'IM_TAGS', text index: 4
    Rectangle (352,150 207x33), text list: 'IM_TAGS', text index: 5
    Rectangle (352,186 207x33), text list: 'IM_TAGS', text index: 6
    Rectangle (352,222 207x33), text list: 'IM_TAGS', text index: 7
    Rectangle (352,258 207x33), text list: 'IM_TAGS', text index: 8
    Rectangle (352,294 207x33), text list: 'IM_TAGS', text index: 9
    Rectangle (562,42 230x33)
    Button (566,46 105x25), colour toggle: GVL.XV03KV209_TSTOI
        OnMouseClick: execute { GVL.TSTOI := 3; }
    Button (683,46 105x25), colour toggle: GVL.XV04KV210_TSTOI
        OnMouseClick: execute { GVL.TSTOI := 4; }
    Rectangle (562,78 230x33)
    Button (566,82 105x25), colour toggle: GVL.MV01KM00_TSTOI
        OnMouseClick: execute { GVL.TSTOI := 5; }
    Rectangle (562,114 230x33)
    Button (566,118 105x25), colour toggle: GVL.M01UZ01_TSTOI
        OnMouseClick: execute { GVL.TSTOI := 6; }
    Rectangle (562,150 230x33)
    Button (566,154 105x25), colour toggle: GVL.M03UZ03_TSTOI
        OnMouseClick: execute { GVL.TSTOI := 7; }
    Rectangle (562,186 230x33)
    Button (566,190 105x25), colour toggle: GVL.M02UZ02_TSTOI
        OnMouseClick: execute { GVL.TSTOI := 8; }
    Rectangle (562,222 230x33)
    Button (566,226 105x25), colour toggle: GVL.M05UZ05_TSTOI
        OnMouseClick: execute { GVL.TSTOI := 9; }
    Rectangle (562,258 230x33)
    Button (566,262 105x25), colour toggle: GVL.M06UZ06_TSTOI
        OnMouseClick: execute { GVL.TSTOI := 10; }
    Rectangle (562,294 230x33)
    Button (566,298 105x25), colour toggle: GVL.M07KM07_TSTOI
        OnMouseClick: execute { GVL.TSTOI := 11; }
    Image (676,346 105x47), image: VisuSymbols.Symbols.ArrowBoldRight
        OnMouseClick: FrameSelectionChange Selection=Selection=-1, GlobSel=IndExpr=5, AssignDir=Main.GenElemInst_39, AssignType=Directly, SelType=Globally
END_VISUALIZATION

// Device/Application/Main
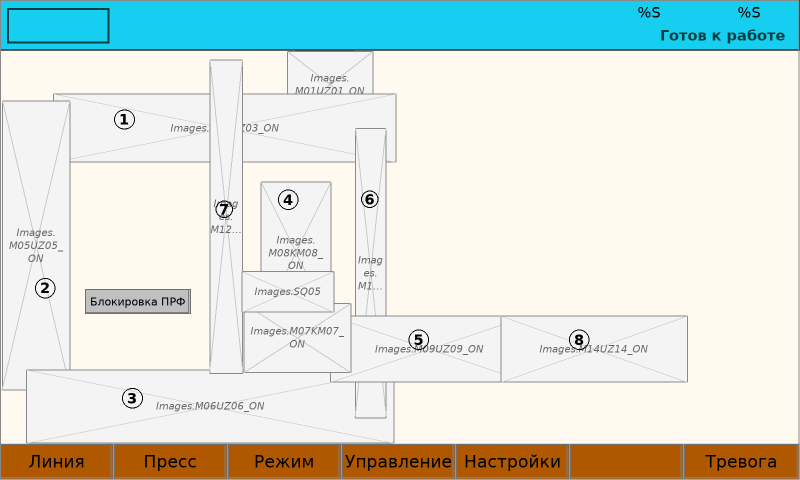
VISUALIZATION Main  // 800x480
    Frame (0,51 800x392)
        shows MAIN_FRAME()
        shows SETTINGS_FRAME()
        shows PRF_FRAME()
        shows ALARM_FRAME()
        shows TEST_FRAME_1()
        shows TEST_FRAME_2()
        shows MANUAL_FRAME_1()
        shows MANUAL_FRAME_2()
        shows MANUAL_FRAME_3()
    Rectangle (0,0 800x50)
    Rectangle (599,0 100x25), "%S", text variable: GVL.PLC_DATE
    Rectangle (699,0 100x25), "%S", text variable: GVL.PLC_TIME
    Button (0,444 113x35), "Линия"
        OnMouseClick: FrameSelectionChange Selection=SelectedFrame=34685d7a-e9ae-4619-9cf1-b28bdaee1b0c, GlobSel=AssignType=Directly, SelType=Locally
    Button (114,444 113x35), "Пресс"
        OnMouseClick: FrameSelectionChange Selection=SelectedFrame=34685d7a-e9ae-4619-9cf1-b28bdaee1b0c, Selection=2, GlobSel=AssignType=Directly, SelType=Locally
    Button (228,444 113x35), "Режим"
        OnMouseClick:  Dialog=MODE_FRAME, OpenModal=True, PositionX=228, PositionY=336
    Button (342,444 113x35), "Управление"
        OnMouseClick: FrameSelectionChange Selection=SelectedFrame=34685d7a-e9ae-4619-9cf1-b28bdaee1b0c, Selection=6, GlobSel=AssignType=Directly, SelType=Locally
    Button (456,444 113x35), "Настройки"
        OnMouseClick: FrameSelectionChange Selection=SelectedFrame=34685d7a-e9ae-4619-9cf1-b28bdaee1b0c, Selection=1, GlobSel=AssignType=Directly, SelType=Locally
    Button (570,444 113x35)
    Button (684,444 115x35), "Тревога"
        OnMouseClick: FrameSelectionChange Selection=SelectedFrame=34685d7a-e9ae-4619-9cf1-b28bdaee1b0c, Selection=3, GlobSel=AssignType=Directly, SelType=Locally
    Textfield (7,8 102x35), text list: 'Mode', text index: GVL.LRF_MODE
    Textfield (170,0 427x50), text list: 'IM', text index: GVL.TSTOI
    Textfield (657,28 129x15), "Готов к работе", invisible if: NOT GVL.LRFRDYSTS
END_VISUALIZATION

// Device/Application/MAIN_FRAME
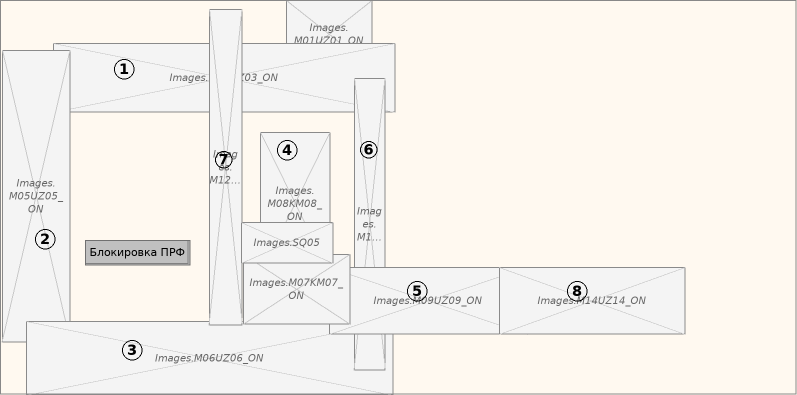
VISUALIZATION MAIN_FRAME  // 797x395, background image Images.Main
    Image (292,-1 63x19), invisible if: NOT GVL.A3_DI_KV301, image: Images.RUN-PRES
    Image (286,0 86x68), invisible if: NOT GVL.A1_DI_MV01KM00_ON, image: Images.MV01KM00_ON
    Image (286,0 86x68), invisible if: GVL.A2_DI_SQ01, image: Images.SQ01
    Image (286,0 86x68), invisible if: NOT GVL.A1_DI_M01UZ01_ON, image: Images.M01UZ01_ON
    Image (286,49 79x40), invisible if: NOT GVL.A1_DI_M04KM04_ON, image: Images.M04KM04_ON
    Image (286,49 79x40), invisible if: NOT GVL.A2_DI_SQ02, image: Images.SQ02
    Image (53,43 342x69), invisible if: NOT GVL.A1_DI_M03UZ03_ON, image: Images.M03UZ03_ON
    Image (2,50 68x292), invisible if: NOT GVL.A1_DI_M05UZ05_ON, image: Images.M05UZ05_ON
    Image (26,321 367x74), invisible if: NOT GVL.A1_DI_M06UZ06_ON, image: Images.M06UZ06_ON
    Image (209,9 33x316), invisible if: NOT GVL.A2_DI_M12KM12_ON, image: Images.M12KM12_ON
    Image (354,78 31x292), invisible if: NOT GVL.A2_DI_M11KM11_ON, image: Images.M11KM11_ON
    Image (260,132 70x143), invisible if: NOT GVL.A1_DI_M08KM08_ON, image: Images.M08KM08_ON
    Image (329,267 198x67), invisible if: NOT GVL.A2_DI_M09UZ09_ON, image: Images.M09UZ09_ON
    Image (499,267 186x67), invisible if: NOT GVL.A2_DI_M14UZ14_ON, image: Images.M14UZ14_ON
    Image (243,254 107x70), invisible if: NOT GVL.A1_DI_M07KM07_ON, image: Images.M07KM07_ON
    Image (241,222 92x41), invisible if: NOT GVL.A2_DI_SQ04, image: Images.SQ04
    Image (241,222 92x41), invisible if: NOT GVL.A2_DI_SQ05, image: Images.SQ05
    Ellipse (114,59 20x20), "1"
    Ellipse (35,229 20x20), "2"
    Ellipse (122,340 20x20), "3"
    Ellipse (277,140 20x20), "4"
    Ellipse (407,281 20x20), "5"
    Ellipse (567,281 20x20), "8"
    Ellipse (360,141 17x17), "6"
    Ellipse (215,151 17x17), "7"
    Button (85,240 105x25), "Блокировка ПРФ", colour toggle: Motors.A2_DI_SQ08_KEEP
        OnMouseClick:  ToggleVariable=Motors.A2_DI_SQ08_KEEP
END_VISUALIZATION

